LIN {X 0,Y 467.847,Z 259.021,A -85,B 0,C 180,E1 -7562.584,E2 -7562.584} C_VEL
LIN {X 0,Y 467.734,Z 259.031,A -85,B 0,C 180,E1 -7566.039,E2 -7566.039} C_VEL
LIN {X 0,Y 467.669,Z 259.046,A -85,B 0,C 180,E1 -7568.644,E2 -7568.644} C_VEL
LIN {X 0,Y 467.664,Z 259.043,A -85,B 0,C 180,E1 -7572.37,E2 -7572.37} C_VEL
LIN {X 0,Y 467.64,Z 259.045,A -85,B 0,C 180,E1 -7575.887,E2 -7575.887} C_VEL
LIN {X 0,Y 467.612,Z 259.05,A -85,B 0,C 180,E1 -7579.309,E2 -7579.309} C_VEL
LIN {X 0,Y 467.528,Z 259.059,A -85,B 0,C 180,E1 -7582.075,E2 -7582.075} C_VEL
LIN {X 0,Y 467.585,Z 259.054,A -85,B 0,C 180,E1 -7584.89,E2 -7584.89} C_VEL
LIN {X 0,Y 467.572,Z 259.059,A -85,B 0,C 180,E1 -7587.773,E2 -7587.773} C_VEL
LIN {X 0,Y 467.563,Z 259.06,A -85,B 0,C 180,E1 -7591.047,E2 -7591.047} C_VEL
LIN {X 0,Y 467.582,Z 259.057,A -85,B 0,C 180,E1 -7594.244,E2 -7594.244} C_VEL
LIN {X 0,Y 467.537,Z 259.064,A -85,B 0,C 180,E1 -7597.187,E2 -7597.187} C_VEL
LIN {X 0,Y 467.59,Z 259.056,A -85,B 0,C 180,E1 -7600.264,E2 -7600.264} C_VEL
LIN {X 0,Y 467.582,Z 259.054,A -85,B 0,C 180,E1 -7602.569,E2 -7602.569} C_VEL
LIN {X 0,Y 467.561,Z 259.062,A -85,B 0,C 180,E1 -7605.054,E2 -7605.054} C_VEL
LIN {X 0,Y 467.585,Z 259.056,A -85,B 0,C 180,E1 -7607.441,E2 -7607.441} C_VEL
LIN {X 0,Y 467.578,Z 259.057,A -85,B 0,C 180,E1 -7610.857,E2 -7610.857} C_VEL
LIN {X 0,Y 467.576,Z 259.195,A -85,B 0,C 180,E1 -7613.246,E2 -7613.246} C_VEL
LIN {X 0,Y 468.724,Z 265.645,A -85,B 0,C 180,E1 -7616.307,E2 -7616.307} C_VEL
LIN {X 0,Y 468.772,Z 270.316,A -85,B 0,C 180,E1 -7618.351,E2 -7618.351} C_VEL
LIN {X 0,Y 468.223,Z 278.68,A -85,B 0,C 180,E1 -7621.784,E2 -7621.784} C_VEL
LIN {X 0,Y 467.766,Z 287.187,A -85,B 0,C 180,E1 -7625.123,E2 -7625.123} C_VEL
LIN {X 0,Y 467.482,Z 294.551,A -85,B 0,C 180,E1 -7627.925,E2 -7627.925} C_VEL
LIN {X 0,Y 467.187,Z 304.438,A -85,B 0,C 180,E1 -7631.586,E2 -7631.586} C_VEL
LIN {X 0,Y 466.983,Z 313.335,A -85,B 0,C 180,E1 -7634.792,E2 -7634.792} C_VEL
LIN {X 0,Y 466.835,Z 321.809,A -85,B 0,C 180,E1 -7637.807,E2 -7637.807} C_VEL
LIN {X 0,Y 468.169,Z 334.234,A -85,B 0,C 180,E1 -7638.248,E2 -7638.248} C_VEL
LIN {X 0,Y 468.576,Z 341.804,A -85,B 0,C 180,E1 -7638.606,E2 -7638.606} C_VEL
LIN {X 0,Y 468.272,Z 351.549,A -85,B 0,C 180,E1 -7639.188,E2 -7639.188} C_VEL
LIN {X 0,Y 467.927,Z 360.068,A -85,B 0,C 180,E1 -7639.837,E2 -7639.837} C_VEL
LIN {X 0,Y 467.577,Z 368.103,A -85,B 0,C 180,E1 -7640.594,E2 -7640.594} C_VEL
LIN {X 0,Y 467.357,Z 374.752,A -85,B 0,C 180,E1 -7641.352,E2 -7641.352} C_VEL
LIN {X 0,Y 467.106,Z 381.074,A -85,B 0,C 180,E1 -7642.219,E2 -7642.219} C_VEL
LIN {X 0,Y 466.94,Z 386.332,A -85,B 0,C 180,E1 -7643.085,E2 -7643.085} C_VEL
LIN {X 0,Y 466.833,Z 390.722,A -85,B 0,C 180,E1 -7643.952,E2 -7643.952} C_VEL
LIN {X 0,Y 466.719,Z 395.908,A -85,B 0,C 180,E1 -7645.25,E2 -7645.25} C_VEL
LIN {X 0,Y 466.757,Z 399.722,A -85,B 0,C 180,E1 -7646.548,E2 -7646.548} C_VEL
LIN {X 0,Y 466.686,Z 401.467,A -85,B 0,C 180,E1 -7647.412,E2 -7647.412} C_VEL
LIN {X 0,Y 466.661,Z 402.717,A -85,B 0,C 180,E1 -7648.275,E2 -7648.275} C_VEL
LIN {X 0,Y 466.62,Z 403.491,A -85,B 0,C 180,E1 -7649.138,E2 -7649.138} C_VEL
LIN {X 0,Y 466.603,Z 403.785,A -85,B 0,C 180,E1 -7650.001,E2 -7650.001} C_VEL
LIN {X 0,Y 466.62,Z 403.487,A -85,B 0,C 180,E1 -7650.864,E2 -7650.864} C_VEL
LIN {X 0,Y 466.661,Z 402.692,A -85,B 0,C 180,E1 -7651.727,E2 -7651.727} C_VEL
LIN {X 0,Y 466.686,Z 401.42,A -85,B 0,C 180,E1 -7652.59,E2 -7652.59} C_VEL
LIN {X 0,Y 466.717,Z 398.486,A -85,B 0,C 180,E1 -7653.887,E2 -7653.887} C_VEL
LIN {X 0,Y 466.719,Z 395.804,A -85,B 0,C 180,E1 -7654.752,E2 -7654.752} C_VEL
LIN {X 0,Y 466.833,Z 392.504,A -85,B 0,C 180,E1 -7655.617,E2 -7655.617} C_VEL
LIN {X 0,Y 466.952,Z 387.176,A -85,B 0,C 180,E1 -7656.725,E2 -7656.725} C_VEL
LIN {X 0,Y 467.098,Z 380.806,A -85,B 0,C 180,E1 -7657.784,E2 -7657.784} C_VEL
LIN {X 0,Y 467.415,Z 372.688,A -85,B 0,C 180,E1 -7658.867,E2 -7658.867} C_VEL
LIN {X 0,Y 467.752,Z 363.177,A -85,B 0,C 180,E1 -7659.842,E2 -7659.842} C_VEL
LIN {X 0,Y 468.024,Z 355.279,A -85,B 0,C 180,E1 -7660.492,E2 -7660.492} C_VEL
LIN {X 0,Y 468.309,Z 347.164,A -85,B 0,C 180,E1 -7661.032,E2 -7661.032} C_VEL
LIN {X 0,Y 468.501,Z 338.954,A -85,B 0,C 180,E1 -7661.468,E2 -7661.468} C_VEL
LIN {X 0,Y 467.685,Z 330.12,A -85,B 0,C 180,E1 -7661.845,E2 -7661.845} C_VEL
LIN {X 0,Y 466.831,Z 321.957,A -85,B 0,C 180,E1 -7662.122,E2 -7662.122} C_VEL
LIN {X 0,Y 466.971,Z 313.201,A -85,B 0,C 180,E1 -7665.207,E2 -7665.207} C_VEL
LIN {X 0,Y 467.162,Z 304.206,A -85,B 0,C 180,E1 -7668.418,E2 -7668.418} C_VEL
LIN {X 0,Y 467.393,Z 295.384,A -85,B 0,C 180,E1 -7671.617,E2 -7671.617} C_VEL
LIN {X 0,Y 467.714,Z 286.565,A -85,B 0,C 180,E1 -7674.882,E2 -7674.882} C_VEL
LIN {X 0,Y 468.048,Z 279.032,A -85,B 0,C 180,E1 -7677.742,E2 -7677.742} C_VEL
LIN {X 0,Y 468.398,Z 271.514,A -85,B 0,C 180,E1 -7680.675,E2 -7680.675} C_VEL
LIN {X 0,Y 468.62,Z 265.139,A -85,B 0,C 180,E1 -7683.246,E2 -7683.246} C_VEL
LIN {X 0,Y 467.569,Z 259.058,A -85,B 0,C 180,E1 -7685.889,E2 -7685.889} C_VEL
LIN {X 0,Y 467.568,Z 259.057,A -85,B 0,C 180,E1 -7689.147,E2 -7689.147} C_VEL
LIN {X 0,Y 467.595,Z 259.053,A -85,B 0,C 180,E1 -7692.567,E2 -7692.567} C_VEL
LIN {X 0,Y 467.574,Z 259.054,A -85,B 0,C 180,E1 -7695.053,E2 -7695.053} C_VEL
LIN {X 0,Y 467.598,Z 259.053,A -85,B 0,C 180,E1 -7697.44,E2 -7697.44} C_VEL
LIN {X 0,Y 467.568,Z 259.056,A -85,B 0,C 180,E1 -7700.853,E2 -7700.853} C_VEL
LIN {X 0,Y 467.566,Z 259.058,A -85,B 0,C 180,E1 -7704.261,E2 -7704.261} C_VEL
LIN {X 0,Y 467.59,Z 259.055,A -85,B 0,C 180,E1 -7707.321,E2 -7707.321} C_VEL
LIN {X 0,Y 467.578,Z 259.055,A -85,B 0,C 180,E1 -7710.667,E2 -7710.667} C_VEL
LIN {X 0,Y 467.622,Z 259.051,A -85,B 0,C 180,E1 -7713.199,E2 -7713.199} C_VEL
LIN {X 0,Y 467.6,Z 259.052,A -85,B 0,C 180,E1 -7716.468,E2 -7716.468} C_VEL
LIN {X 0,Y 467.631,Z 259.048,A -85,B 0,C 180,E1 -7719.776,E2 -7719.776} C_VEL
LIN {X 0,Y 467.606,Z 259.051,A -85,B 0,C 180,E1 -7722.505,E2 -7722.505} C_VEL
LIN {X 0,Y 467.613,Z 259.052,A -85,B 0,C 180,E1 -7725.195,E2 -7725.195} C_VEL
LIN {X 0,Y 467.664,Z 259.044,A -85,B 0,C 180,E1 -7727.853,E2 -7727.853} C_VEL
LIN {X 0,Y 467.676,Z 259.043,A -85,B 0,C 180,E1 -7731.356,E2 -7731.356} C_VEL
LIN {X 0,Y 467.74,Z 259.035,A -85,B 0,C 180,E1 -7733.961,E2 -7733.961} C_VEL
LIN {X 0,Y 467.865,Z 259.019,A -85,B 0,C 180,E1 -7737.416,E2 -7737.416} C_VEL
LIN {X 0,Y 467.888,Z 259.017,A -85,B 0,C 180,E1 -7739.998,E2 -7739.998} C_VEL
LIN {X 0,Y 467.865,Z 259.021,A -85,B 0,C 180,E1 -7742.581,E2 -7742.581} C_VEL
LIN {X 0,Y 467.748,Z 259.035,A -85,B 0,C 180,E1 -7746.036,E2 -7746.036} C_VEL
LIN {X 0,Y 467.685,Z 259.043,A -85,B 0,C 180,E1 -7748.641,E2 -7748.641} C_VEL
LIN {X 0,Y 467.659,Z 259.048,A -85,B 0,C 180,E1 -7752.144,E2 -7752.144} C_VEL
LIN {X 0,Y 467.641,Z 259.048,A -85,B 0,C 180,E1 -7755.693,E2 -7755.693} C_VEL
LIN {X 0,Y 467.618,Z 259.05,A -85,B 0,C 180,E1 -7758.762,E2 -7758.762} C_VEL
LIN {X 0,Y 467.58,Z 259.055,A -85,B 0,C 180,E1 -7761.266,E2 -7761.266} C_VEL
LIN {X 0,Y 467.572,Z 259.057,A -85,B 0,C 180,E1 -7763.941,E2 -7763.941} C_VEL
LIN {X 0,Y 467.614,Z 259.049,A -85,B 0,C 180,E1 -7766.798,E2 -7766.798} C_VEL
LIN {X 0,Y 467.551,Z 259.06,A -85,B 0,C 180,E1 -7769.736,E2 -7769.736} C_VEL
LIN {X 0,Y 467.58,Z 259.054,A -85,B 0,C 180,E1 -7772.756,E2 -7772.756} C_VEL
LIN {X 0,Y 467.551,Z 259.059,A -85,B 0,C 180,E1 -7775.887,E2 -7775.887} C_VEL
LIN {X 0,Y 467.608,Z 259.052,A -85,B 0,C 180,E1 -7779.139,E2 -7779.139} C_VEL
LIN {X 0,Y 467.611,Z 259.051,A -85,B 0,C 180,E1 -7782.569,E2 -7782.569} C_VEL
LIN {X 0,Y 467.565,Z 259.056,A -85,B 0,C 180,E1 -7786.174,E2 -7786.174} C_VEL
LIN {X 0,Y 467.581,Z 259.057,A -85,B 0,C 180,E1 -7788.719,E2 -7788.719} C_VEL
LIN {X 0,Y 467.568,Z 259.058,A -85,B 0,C 180,E1 -7791.404,E2 -7791.404} C_VEL
LIN {X 0,Y 467.552,Z 259.057,A -85,B 0,C 180,E1 -7794.258,E2 -7794.258} C_VEL
LIN {X 0,Y 467.569,Z 259.058,A -85,B 0,C 180,E1 -7797.319,E2 -7797.319} C_VEL
LIN {X 0,Y 467.564,Z 259.059,A -85,B 0,C 180,E1 -7800.663,E2 -7800.663} C_VEL
LIN {X 0,Y 467.613,Z 259.051,A -85,B 0,C 180,E1 -7803.198,E2 -7803.198} C_VEL
LIN {X 0,Y 467.582,Z 259.056,A -85,B 0,C 180,E1 -7806.465,E2 -7806.465} C_VEL
LIN {X 0,Y 467.603,Z 259.052,A -85,B 0,C 180,E1 -7809.775,E2 -7809.775} C_VEL
LIN {X 0,Y 467.545,Z 259.059,A -85,B 0,C 180,E1 -7811.629,E2 -7811.629} C_VEL
LIN {X 0,Y 467.186,Z 259.106,A -85,B 0,C 180,E1 -7814.306,E2 -7814.306} C_VEL
LIN {X 0,Y 467.136,Z 260.347,A -85,B 0,C 180,E1 -7815.376,E2 -7815.376} C_VEL
LIN {X 0,Y 466.444,Z 261.32,A -85,B 0,C 180,E1 -7816.087,E2 -7816.087} C_VEL
LIN {X 0,Y 463.58,Z 263.063,A -85,B 0,C 180,E1 -7817.238,E2 -7817.238} C_VEL
LIN {X 0,Y 461.159,Z 264.477,A -85,B 0,C 180,E1 -7818.166,E2 -7818.166} C_VEL
LIN {X 0,Y 460.102,Z 265.496,A -85,B 0,C 180,E1 -7818.884,E2 -7818.884} C_VEL
LIN {X 0,Y 460.005,Z 265.819,A -85,B 0,C 180,E1 -7819.127,E2 -7819.127} C_VEL
LIN {X 0,Y 459.965,Z 269.626,A -85,B 0,C 180,E1 -7822.095,E2 -7822.095} C_VEL
LIN {X 0,Y 459.987,Z 271.938,A -85,B 0,C 180,E1 -7823.859,E2 -7823.859} C_VEL
LIN {X 0,Y 459.964,Z 275.389,A -85,B 0,C 180,E1 -7826.495,E2 -7826.495} C_VEL
LIN {X 0,Y 459.636,Z 280.076,A -85,B 0,C 180,E1 -7829.999,E2 -7829.999} C_VEL
LIN {X 0,Y 459.646,Z 282.543,A -85,B 0,C 180,E1 -7831.833,E2 -7831.833} C_VEL
LIN {X 0,Y 461.767,Z 294.466,A -85,B 0,C 180,E1 -7832.343,E2 -7832.343} C_VEL
LIN {X 0,Y 461.645,Z 302.062,A -85,B 0,C 180,E1 -7832.726,E2 -7832.726} C_VEL
LIN {X 0,Y 461.4,Z 310.62,A -85,B 0,C 180,E1 -7833.273,E2 -7833.273} C_VEL
LIN {X 0,Y 461.077,Z 318.847,A -85,B 0,C 180,E1 -7833.932,E2 -7833.932} C_VEL
LIN {X 0,Y 460.768,Z 326.642,A -85,B 0,C 180,E1 -7834.701,E2 -7834.701} C_VEL
LIN {X 0,Y 460.59,Z 333.057,A -85,B 0,C 180,E1 -7835.471,E2 -7835.471} C_VEL
LIN {X 0,Y 460.357,Z 338.967,A -85,B 0,C 180,E1 -7836.319,E2 -7836.319} C_VEL
LIN {X 0,Y 460.201,Z 344.276,A -85,B 0,C 180,E1 -7837.237,E2 -7837.237} C_VEL
LIN {X 0,Y 459.932,Z 349.496,A -85,B 0,C 180,E1 -7838.346,E2 -7838.346} C_VEL
LIN {X 0,Y 459.757,Z 354.317,A -85,B 0,C 180,E1 -7839.679,E2 -7839.679} C_VEL
LIN {X 0,Y 459.698,Z 356.67,A -85,B 0,C 180,E1 -7840.57,E2 -7840.57} C_VEL
LIN {X 0,Y 459.63,Z 359.185,A -85,B 0,C 180,E1 -7841.89,E2 -7841.89} C_VEL
LIN {X 0,Y 459.534,Z 360.484,A -85,B 0,C 180,E1 -7843.261,E2 -7843.261} C_VEL
LIN {X 0,Y 459.507,Z 360.759,A -85,B 0,C 180,E1 -7844.164,E2 -7844.164} C_VEL
LIN {X 0,Y 459.581,Z 360.016,A -85,B 0,C 180,E1 -7845.558,E2 -7845.558} C_VEL
LIN {X 0,Y 459.654,Z 358.169,A -85,B 0,C 180,E1 -7846.887,E2 -7846.887} C_VEL
LIN {X 0,Y 459.781,Z 355.119,A -85,B 0,C 180,E1 -7848.225,E2 -7848.225} C_VEL
LIN {X 0,Y 460.03,Z 350.431,A -85,B 0,C 180,E1 -7849.638,E2 -7849.638} C_VEL
LIN {X 0,Y 460.2,Z 345.355,A -85,B 0,C 180,E1 -7850.767,E2 -7850.767} C_VEL
LIN {X 0,Y 460.429,Z 340.034,A -85,B 0,C 180,E1 -7851.724,E2 -7851.724} C_VEL
LIN {X 0,Y 460.7,Z 333.714,A -85,B 0,C 180,E1 -7852.654,E2 -7852.654} C_VEL
LIN {X 0,Y 460.98,Z 326.74,A -85,B 0,C 180,E1 -7853.499,E2 -7853.499} C_VEL
LIN {X 0,Y 461.303,Z 318.786,A -85,B 0,C 180,E1 -7854.288,E2 -7854.288} C_VEL
LIN {X 0,Y 461.701,Z 310.029,A -85,B 0,C 180,E1 -7854.985,E2 -7854.985} C_VEL
LIN {X 0,Y 462.023,Z 299.473,A -85,B 0,C 180,E1 -7855.639,E2 -7855.639} C_VEL
LIN {X 0,Y 461.889,Z 294.564,A -85,B 0,C 180,E1 -7855.875,E2 -7855.875} C_VEL
LIN {X 0,Y 460.037,Z 284.59,A -85,B 0,C 180,E1 -7856.316,E2 -7856.316} C_VEL
LIN {X 0,Y 459.668,Z 282.744,A -85,B 0,C 180,E1 -7856.395,E2 -7856.395} C_VEL
LIN {X 0,Y 459.727,Z 278.823,A -85,B 0,C 180,E1 -7859.386,E2 -7859.386} C_VEL
LIN {X 0,Y 459.793,Z 275.013,A -85,B 0,C 180,E1 -7862.341,E2 -7862.341} C_VEL
LIN {X 0,Y 459.887,Z 270.511,A -85,B 0,C 180,E1 -7865.914,E2 -7865.914} C_VEL
LIN {X 0,Y 459.949,Z 266.915,A -85,B 0,C 180,E1 -7868.809,E2 -7868.809} C_VEL
LIN {X 0,Y 460.094,Z 262.754,A -85,B 0,C 180,E1 -7872.228,E2 -7872.228} C_VEL
LIN {X 0,Y 460.179,Z 259.979,A -85,B 0,C 180,E1 -7874.628,E2 -7874.628} C_VEL
LIN {X 0,Y 460.412,Z 259.944,A -85,B 0,C 180,E1 -7877.111,E2 -7877.111} C_VEL
LIN {X 0,Y 460.557,Z 259.928,A -85,B 0,C 180,E1 -7880.143,E2 -7880.143} C_VEL
LIN {X 0,Y 460.461,Z 259.941,A -85,B 0,C 180,E1 -7883.472,E2 -7883.472} C_VEL
LIN {X 0,Y 460.51,Z 259.934,A -85,B 0,C 180,E1 -7886.676,E2 -7886.676} C_VEL
LIN {X 0,Y 460.491,Z 259.936,A -85,B 0,C 180,E1 -7889.761,E2 -7889.761} C_VEL
LIN {X 0,Y 460.56,Z 259.927,A -85,B 0,C 180,E1 -7892.758,E2 -7892.758} C_VEL
LIN {X 0,Y 460.52,Z 259.932,A -85,B 0,C 180,E1 -7895.669,E2 -7895.669} C_VEL
LIN {X 0,Y 460.504,Z 259.936,A -85,B 0,C 180,E1 -7898.579,E2 -7898.579} C_VEL
LIN {X 0,Y 460.575,Z 259.927,A -85,B 0,C 180,E1 -7901.312,E2 -7901.312} C_VEL
LIN {X 0,Y 460.588,Z 259.924,A -85,B 0,C 180,E1 -7904.06,E2 -7904.06} C_VEL
LIN {X 0,Y 460.615,Z 259.922,A -85,B 0,C 180,E1 -7907.668,E2 -7907.668} C_VEL
LIN {X 0,Y 460.615,Z 259.925,A -85,B 0,C 180,E1 -7911.225,E2 -7911.225} C_VEL
LIN {X 0,Y 460.671,Z 259.911,A -85,B 0,C 180,E1 -7913.871,E2 -7913.871} C_VEL
LIN {X 0,Y 460.815,Z 259.898,A -85,B 0,C 180,E1 -7917.379,E2 -7917.379} C_VEL
LIN {X 0,Y 460.84,Z 259.892,A -85,B 0,C 180,E1 -7920.002,E2 -7920.002} C_VEL
LIN {X 0,Y 460.788,Z 259.9,A -85,B 0,C 180,E1 -7922.624,E2 -7922.624} C_VEL
LIN {X 0,Y 460.7,Z 259.906,A -85,B 0,C 180,E1 -7926.131,E2 -7926.131} C_VEL
LIN {X 0,Y 460.616,Z 259.923,A -85,B 0,C 180,E1 -7928.778,E2 -7928.778} C_VEL
LIN {X 0,Y 460.625,Z 259.919,A -85,B 0,C 180,E1 -7932.458,E2 -7932.458} C_VEL
LIN {X 0,Y 460.591,Z 259.924,A -85,B 0,C 180,E1 -7935.999,E2 -7935.999} C_VEL
LIN {X 0,Y 460.559,Z 259.931,A -85,B 0,C 180,E1 -7939.617,E2 -7939.617} C_VEL
LIN {X 0,Y 460.504,Z 259.935,A -85,B 0,C 180,E1 -7942.43,E2 -7942.43} C_VEL
LIN {X 0,Y 460.542,Z 259.933,A -85,B 0,C 180,E1 -7945.799,E2 -7945.799} C_VEL
LIN {X 0,Y 460.519,Z 259.934,A -85,B 0,C 180,E1 -7948.236,E2 -7948.236} C_VEL
LIN {X 0,Y 460.516,Z 259.936,A -85,B 0,C 180,E1 -7951.285,E2 -7951.285} C_VEL
LIN {X 0,Y 460.525,Z 259.935,A -85,B 0,C 180,E1 -7954.507,E2 -7954.507} C_VEL
LIN {X 0,Y 460.495,Z 259.937,A -85,B 0,C 180,E1 -7957.625,E2 -7957.625} C_VEL
LIN {X 0,Y 460.553,Z 259.933,A -85,B 0,C 180,E1 -7960.273,E2 -7960.273} C_VEL
LIN {X 0,Y 460.494,Z 259.941,A -85,B 0,C 180,E1 -7963.377,E2 -7963.377} C_VEL
LIN {X 0,Y 460.494,Z 259.938,A -85,B 0,C 180,E1 -7966.626,E2 -7966.626} C_VEL
LIN {X 0,Y 460.538,Z 259.934,A -85,B 0,C 180,E1 -7969.732,E2 -7969.732} C_VEL
LIN {X 0,Y 460.508,Z 259.977,A -85,B 0,C 180,E1 -7972.929,E2 -7972.929} C_VEL
LIN {X 0,Y 461.544,Z 265.68,A -85,B 0,C 180,E1 -7975.71,E2 -7975.71} C_VEL
LIN {X 0,Y 461.861,Z 269.21,A -85,B 0,C 180,E1 -7977.325,E2 -7977.325} C_VEL
LIN {X 0,Y 461.446,Z 276.023,A -85,B 0,C 180,E1 -7980.243,E2 -7980.243} C_VEL
LIN {X 0,Y 460.978,Z 283.444,A -85,B 0,C 180,E1 -7983.274,E2 -7983.274} C_VEL
LIN {X 0,Y 460.581,Z 291.954,A -85,B 0,C 180,E1 -7986.627,E2 -7986.627} C_VEL
LIN {X 0,Y 460.207,Z 300.556,A -85,B 0,C 180,E1 -7989.905,E2 -7989.905} C_VEL
LIN {X 0,Y 459.993,Z 309.209,A -85,B 0,C 180,E1 -7993.126,E2 -7993.126} C_VEL
LIN {X 0,Y 459.8,Z 317.907,A -85,B 0,C 180,E1 -7996.297,E2 -7996.297} C_VEL
LIN {X 0,Y 459.762,Z 321.484,A -85,B 0,C 180,E1 -7997.588,E2 -7997.588} C_VEL
LIN {X 0,Y 461.195,Z 334.661,A -85,B 0,C 180,E1 -7998.082,E2 -7998.082} C_VEL
LIN {X 0,Y 461.623,Z 342.117,A -85,B 0,C 180,E1 -7998.448,E2 -7998.448} C_VEL
LIN {X 0,Y 461.308,Z 351.464,A -85,B 0,C 180,E1 -7999.023,E2 -7999.023} C_VEL
LIN {X 0,Y 460.935,Z 359.927,A -85,B 0,C 180,E1 -7999.681,E2 -7999.681} C_VEL
LIN {X 0,Y 460.564,Z 367.92,A -85,B 0,C 180,E1 -8000.449,E2 -8000.449} C_VEL
LIN {X 0,Y 460.306,Z 374.536,A -85,B 0,C 180,E1 -8001.219,E2 -8001.219} C_VEL
LIN {X 0,Y 460.062,Z 380.831,A -85,B 0,C 180,E1 -8002.099,E2 -8002.099} C_VEL
LIN {X 0,Y 459.873,Z 386.07,A -85,B 0,C 180,E1 -8002.979,E2 -8002.979} C_VEL
LIN {X 0,Y 459.742,Z 390.446,A -85,B 0,C 180,E1 -8003.858,E2 -8003.858} C_VEL
LIN {X 0,Y 459.65,Z 395.622,A -85,B 0,C 180,E1 -8005.177,E2 -8005.177} C_VEL
LIN {X 0,Y 459.651,Z 399.424,A -85,B 0,C 180,E1 -8006.495,E2 -8006.495} C_VEL
LIN {X 0,Y 459.609,Z 401.161,A -85,B 0,C 180,E1 -8007.372,E2 -8007.372} C_VEL
LIN {X 0,Y 459.57,Z 402.401,A -85,B 0,C 180,E1 -8008.248,E2 -8008.248} C_VEL
LIN {X 0,Y 459.553,Z 403.167,A -85,B 0,C 180,E1 -8009.125,E2 -8009.125} C_VEL
LIN {X 0,Y 459.534,Z 403.455,A -85,B 0,C 180,E1 -8010.001,E2 -8010.001} C_VEL
LIN {X 0,Y 459.553,Z 403.154,A -85,B 0,C 180,E1 -8010.877,E2 -8010.877} C_VEL
LIN {X 0,Y 459.571,Z 402.348,A -85,B 0,C 180,E1 -8011.754,E2 -8011.754} C_VEL
LIN {X 0,Y 459.609,Z 401.066,A -85,B 0,C 180,E1 -8012.63,E2 -8012.63} C_VEL
LIN {X 0,Y 459.611,Z 398.119,A -85,B 0,C 180,E1 -8013.947,E2 -8013.947} C_VEL
LIN {X 0,Y 459.651,Z 395.427,A -85,B 0,C 180,E1 -8014.825,E2 -8014.825} C_VEL
LIN {X 0,Y 459.732,Z 392.113,A -85,B 0,C 180,E1 -8015.704,E2 -8015.704} C_VEL
LIN {X 0,Y 459.883,Z 387.077,A -85,B 0,C 180,E1 -8016.772,E2 -8016.772} C_VEL
LIN {X 0,Y 459.993,Z 381.813,A -85,B 0,C 180,E1 -8017.684,E2 -8017.684} C_VEL
LIN {X 0,Y 460.224,Z 375.68,A -85,B 0,C 180,E1 -8018.564,E2 -8018.564} C_VEL
LIN {X 0,Y 460.446,Z 369.243,A -85,B 0,C 180,E1 -8019.334,E2 -8019.334} C_VEL
LIN {X 0,Y 460.786,Z 361.452,A -85,B 0,C 180,E1 -8020.103,E2 -8020.103} C_VEL
LIN {X 0,Y 461.023,Z 354.747,A -85,B 0,C 180,E1 -8020.653,E2 -8020.653} C_VEL
LIN {X 0,Y 461.314,Z 346.571,A -85,B 0,C 180,E1 -8021.202,E2 -8021.202} C_VEL
LIN {X 0,Y 461.434,Z 338.943,A -85,B 0,C 180,E1 -8021.614,E2 -8021.614} C_VEL
LIN {X 0,Y 460.547,Z 329.166,A -85,B 0,C 180,E1 -8022.033,E2 -8022.033} C_VEL
LIN {X 0,Y 459.752,Z 321.703,A -85,B 0,C 180,E1 -8022.275,E2 -8022.275} C_VEL
LIN {X 0,Y 459.921,Z 312.172,A -85,B 0,C 180,E1 -8025.698,E2 -8025.698} C_VEL
LIN {X 0,Y 460.115,Z 302.765,A -85,B 0,C 180,E1 -8029.126,E2 -8029.126} C_VEL
LIN {X 0,Y 460.408,Z 293.823,A -85,B 0,C 180,E1 -8032.435,E2 -8032.435} C_VEL
LIN {X 0,Y 460.773,Z 284.821,A -85,B 0,C 180,E1 -8035.853,E2 -8035.853} C_VEL
LIN {X 0,Y 461.18,Z 276.269,A -85,B 0,C 180,E1 -8039.187,E2 -8039.187} C_VEL
LIN {X 0,Y 461.566,Z 268.781,A -85,B 0,C 180,E1 -8042.204,E2 -8042.204} C_VEL
LIN {X 0,Y 461.442,Z 265.042,A -85,B 0,C 180,E1 -8043.775,E2 -8043.775} C_VEL
LIN {X 0,Y 460.507,Z 259.938,A -85,B 0,C 180,E1 -8046.089,E2 -8046.089} C_VEL
LIN {X 0,Y 460.542,Z 259.932,A -85,B 0,C 180,E1 -8048.896,E2 -8048.896} C_VEL
LIN {X 0,Y 460.531,Z 259.935,A -85,B 0,C 180,E1 -8052.182,E2 -8052.182} C_VEL
LIN {X 0,Y 460.521,Z 259.934,A -85,B 0,C 180,E1 -8055.411,E2 -8055.411} C_VEL
LIN {X 0,Y 460.54,Z 259.932,A -85,B 0,C 180,E1 -8058.398,E2 -8058.398} C_VEL
LIN {X 0,Y 460.526,Z 259.934,A -85,B 0,C 180,E1 -8061.266,E2 -8061.266} C_VEL
LIN {X 0,Y 460.517,Z 259.934,A -85,B 0,C 180,E1 -8064.554,E2 -8064.554} C_VEL
LIN {X 0,Y 460.54,Z 259.933,A -85,B 0,C 180,E1 -8067.715,E2 -8067.715} C_VEL
LIN {X 0,Y 460.548,Z 259.931,A -85,B 0,C 180,E1 -8070.768,E2 -8070.768} C_VEL
LIN {X 0,Y 460.565,Z 259.93,A -85,B 0,C 180,E1 -8073.734,E2 -8073.734} C_VEL
LIN {X 0,Y 460.553,Z 259.93,A -85,B 0,C 180,E1 -8076.623,E2 -8076.623} C_VEL
LIN {X 0,Y 460.56,Z 259.931,A -85,B 0,C 180,E1 -8079.452,E2 -8079.452} C_VEL
LIN {X 0,Y 460.557,Z 259.928,A -85,B 0,C 180,E1 -8082.229,E2 -8082.229} C_VEL
LIN {X 0,Y 460.572,Z 259.93,A -85,B 0,C 180,E1 -8084.964,E2 -8084.964} C_VEL
LIN {X 0,Y 460.617,Z 259.923,A -85,B 0,C 180,E1 -8088.558,E2 -8088.558} C_VEL
LIN {X 0,Y 460.626,Z 259.922,A -85,B 0,C 180,E1 -8091.222,E2 -8091.222} C_VEL
LIN {X 0,Y 460.705,Z 259.911,A -85,B 0,C 180,E1 -8093.869,E2 -8093.869} C_VEL
LIN {X 0,Y 460.806,Z 259.898,A -85,B 0,C 180,E1 -8097.376,E2 -8097.376} C_VEL
LIN {X 0,Y 460.858,Z 259.892,A -85,B 0,C 180,E1 -8099.998,E2 -8099.998} C_VEL
LIN {X 0,Y 460.83,Z 259.897,A -85,B 0,C 180,E1 -8102.621,E2 -8102.621} C_VEL
LIN {X 0,Y 460.714,Z 259.912,A -85,B 0,C 180,E1 -8106.128,E2 -8106.128} C_VEL
LIN {X 0,Y 460.632,Z 259.922,A -85,B 0,C 180,E1 -8108.774,E2 -8108.774} C_VEL
LIN {X 0,Y 460.616,Z 259.923,A -85,B 0,C 180,E1 -8112.443,E2 -8112.443} C_VEL
LIN {X 0,Y 460.602,Z 259.926,A -85,B 0,C 180,E1 -8115.995,E2 -8115.995} C_VEL
LIN {X 0,Y 460.572,Z 259.928,A -85,B 0,C 180,E1 -8118.9,E2 -8118.9} C_VEL
LIN {X 0,Y 460.516,Z 259.936,A -85,B 0,C 180,E1 -8121.483,E2 -8121.483} C_VEL
LIN {X 0,Y 460.541,Z 259.932,A -85,B 0,C 180,E1 -8124.33,E2 -8124.33} C_VEL
LIN {X 0,Y 460.577,Z 259.927,A -85,B 0,C 180,E1 -8127.241,E2 -8127.241} C_VEL
LIN {X 0,Y 460.508,Z 259.936,A -85,B 0,C 180,E1 -8130.238,E2 -8130.238} C_VEL
LIN {X 0,Y 460.525,Z 259.935,A -85,B 0,C 180,E1 -8133.323,E2 -8133.323} C_VEL
LIN {X 0,Y 460.473,Z 259.939,A -85,B 0,C 180,E1 -8136.527,E2 -8136.527} C_VEL
LIN {X 0,Y 460.569,Z 259.929,A -85,B 0,C 180,E1 -8139.855,E2 -8139.855} C_VEL
LIN {X 0,Y 460.535,Z 259.933,A -85,B 0,C 180,E1 -8142.902,E2 -8142.902} C_VEL
LIN {X 0,Y 460.515,Z 259.935,A -85,B 0,C 180,E1 -8145.826,E2 -8145.826} C_VEL
LIN {X 0,Y 460.534,Z 259.934,A -85,B 0,C 180,E1 -8148.988,E2 -8148.988} C_VEL
LIN {X 0,Y 460.537,Z 259.934,A -85,B 0,C 180,E1 -8151.267,E2 -8151.267} C_VEL
LIN {X 0,Y 460.502,Z 259.937,A -85,B 0,C 180,E1 -8154.553,E2 -8154.553} C_VEL
LIN {X 0,Y 460.52,Z 259.934,A -85,B 0,C 180,E1 -8157.714,E2 -8157.714} C_VEL
LIN {X 0,Y 460.534,Z 259.935,A -85,B 0,C 180,E1 -8160.768,E2 -8160.768} C_VEL
LIN {X 0,Y 460.553,Z 259.93,A -85,B 0,C 180,E1 -8163.733,E2 -8163.733} C_VEL
LIN {X 0,Y 460.536,Z 259.935,A -85,B 0,C 180,E1 -8166.622,E2 -8166.622} C_VEL
LIN {X 0,Y 460.552,Z 259.93,A -85,B 0,C 180,E1 -8169.452,E2 -8169.452} C_VEL
LIN {X 0,Y 460.377,Z 259.954,A -85,B 0,C 180,E1 -8172.222,E2 -8172.222} C_VEL
LIN {X 0,Y 460.146,Z 259.983,A -85,B 0,C 180,E1 -8174.192,E2 -8174.192} C_VEL
LIN {X 0,Y 460.066,Z 261.03,A -85,B 0,C 180,E1 -8175.357,E2 -8175.357} C_VEL
LIN {X 0,Y 460.137,Z 264.123,A -85,B 0,C 180,E1 -8177.815,E2 -8177.815} C_VEL
LIN {X 0,Y 460.005,Z 265.819,A -85,B 0,C 180,E1 -8179.127,E2 -8179.127} C_VEL
LIN {X 0,Y 459.305,Z 266.814,A -85,B 0,C 180,E1 -8179.847,E2 -8179.847} C_VEL
LIN {X 0,Y 456.424,Z 268.581,A -85,B 0,C 180,E1 -8181.013,E2 -8181.013} C_VEL
LIN {X 0,Y 454.022,Z 270.002,A -85,B 0,C 180,E1 -8181.953,E2 -8181.953} C_VEL
LIN {X 0,Y 453.016,Z 271.021,A -85,B 0,C 180,E1 -8182.681,E2 -8182.681} C_VEL
LIN {X 0,Y 452.946,Z 271.343,A -85,B 0,C 180,E1 -8182.928,E2 -8182.928} C_VEL
LIN {X 0,Y 452.886,Z 275.91,A -85,B 0,C 180,E1 -8186.44,E2 -8186.44} C_VEL
LIN {X 0,Y 452.562,Z 280.628,A -85,B 0,C 180,E1 -8189.999,E2 -8189.999} C_VEL
LIN {X 0,Y 452.579,Z 282.861,A -85,B 0,C 180,E1 -8191.667,E2 -8191.667} C_VEL
LIN {X 0,Y 454.63,Z 294.343,A -85,B 0,C 180,E1 -8192.158,E2 -8192.158} C_VEL
LIN {X 0,Y 454.733,Z 300.061,A -85,B 0,C 180,E1 -8192.435,E2 -8192.435} C_VEL
LIN {X 0,Y 454.425,Z 310.592,A -85,B 0,C 180,E1 -8193.102,E2 -8193.102} C_VEL
LIN {X 0,Y 454.112,Z 318.874,A -85,B 0,C 180,E1 -8193.77,E2 -8193.77} C_VEL
LIN {X 0,Y 453.775,Z 326.722,A -85,B 0,C 180,E1 -8194.551,E2 -8194.551} C_VEL
LIN {X 0,Y 453.57,Z 333.182,A -85,B 0,C 180,E1 -8195.333,E2 -8195.333} C_VEL
LIN {X 0,Y 453.299,Z 339.352,A -85,B 0,C 180,E1 -8196.229,E2 -8196.229} C_VEL
LIN {X 0,Y 453.102,Z 345.643,A -85,B 0,C 180,E1 -8197.351,E2 -8197.351} C_VEL
LIN {X 0,Y 452.845,Z 350.67,A -85,B 0,C 180,E1 -8198.477,E2 -8198.477} C_VEL
LIN {X 0,Y 452.657,Z 355.183,A -85,B 0,C 180,E1 -8199.832,E2 -8199.832} C_VEL
LIN {X 0,Y 452.617,Z 357.476,A -85,B 0,C 180,E1 -8200.737,E2 -8200.737} C_VEL
LIN {X 0,Y 452.545,Z 359.599,A -85,B 0,C 180,E1 -8201.947,E2 -8201.947} C_VEL
LIN {X 0,Y 452.429,Z 360.888,A -85,B 0,C 180,E1 -8203.473,E2 -8203.473} C_VEL
LIN {X 0,Y 452.44,Z 361.022,A -85,B 0,C 180,E1 -8204.39,E2 -8204.39} C_VEL
LIN {X 0,Y 452.492,Z 360.297,A -85,B 0,C 180,E1 -8205.651,E2 -8205.651} C_VEL
LIN {X 0,Y 452.53,Z 359.679,A -85,B 0,C 180,E1 -8206.232,E2 -8206.232} C_VEL
LIN {X 0,Y 452.667,Z 357.212,A -85,B 0,C 180,E1 -8207.622,E2 -8207.622} C_VEL
LIN {X 0,Y 452.831,Z 353.298,A -85,B 0,C 180,E1 -8209.02,E2 -8209.02} C_VEL
LIN {X 0,Y 453.007,Z 349.884,A -85,B 0,C 180,E1 -8209.955,E2 -8209.955} C_VEL
LIN {X 0,Y 453.181,Z 345.676,A -85,B 0,C 180,E1 -8210.895,E2 -8210.895} C_VEL
LIN {X 0,Y 453.415,Z 340.537,A -85,B 0,C 180,E1 -8211.838,E2 -8211.838} C_VEL
LIN {X 0,Y 453.694,Z 334.25,A -85,B 0,C 180,E1 -8212.783,E2 -8212.783} C_VEL
LIN {X 0,Y 453.997,Z 327.583,A -85,B 0,C 180,E1 -8213.611,E2 -8213.611} C_VEL
LIN {X 0,Y 454.333,Z 319.976,A -85,B 0,C 180,E1 -8214.39,E2 -8214.39} C_VEL
LIN {X 0,Y 454.699,Z 312.311,A -85,B 0,C 180,E1 -8215.03,E2 -8215.03} C_VEL
LIN {X 0,Y 455.004,Z 303.475,A -85,B 0,C 180,E1 -8215.624,E2 -8215.624} C_VEL
LIN {X 0,Y 455,Z 295.645,A -85,B 0,C 180,E1 -8216.044,E2 -8216.044} C_VEL
LIN {X 0,Y 453.257,Z 286.337,A -85,B 0,C 180,E1 -8216.479,E2 -8216.479} C_VEL
LIN {X 0,Y 452.596,Z 283.071,A -85,B 0,C 180,E1 -8216.634,E2 -8216.634} C_VEL
LIN {X 0,Y 452.66,Z 278.969,A -85,B 0,C 180,E1 -8219.789,E2 -8219.789} C_VEL
LIN {X 0,Y 452.744,Z 274.813,A -85,B 0,C 180,E1 -8223.049,E2 -8223.049} C_VEL
LIN {X 0,Y 452.819,Z 270.898,A -85,B 0,C 180,E1 -8226.194,E2 -8226.194} C_VEL
LIN {X 0,Y 452.904,Z 266.851,A -85,B 0,C 180,E1 -8229.509,E2 -8229.509} C_VEL
LIN {X 0,Y 453.011,Z 264.005,A -85,B 0,C 180,E1 -8231.873,E2 -8231.873} C_VEL
LIN {X 0,Y 453.113,Z 260.92,A -85,B 0,C 180,E1 -8234.485,E2 -8234.485} C_VEL
LIN {X 0,Y 453.355,Z 260.824,A -85,B 0,C 180,E1 -8236.996,E2 -8236.996} C_VEL
LIN {X 0,Y 453.495,Z 260.811,A -85,B 0,C 180,E1 -8239.407,E2 -8239.407} C_VEL
LIN {X 0,Y 453.458,Z 260.814,A -85,B 0,C 180,E1 -8242.223,E2 -8242.223} C_VEL
LIN {X 0,Y 453.47,Z 260.812,A -85,B 0,C 180,E1 -8245.223,E2 -8245.223} C_VEL
LIN {X 0,Y 453.446,Z 260.814,A -85,B 0,C 180,E1 -8248.476,E2 -8248.476} C_VEL
LIN {X 0,Y 453.519,Z 260.807,A -85,B 0,C 180,E1 -8252.04,E2 -8252.04} C_VEL
LIN {X 0,Y 453.489,Z 260.812,A -85,B 0,C 180,E1 -8255.266,E2 -8255.266} C_VEL
LIN {X 0,Y 453.463,Z 260.815,A -85,B 0,C 180,E1 -8258.416,E2 -8258.416} C_VEL
LIN {X 0,Y 453.506,Z 260.806,A -85,B 0,C 180,E1 -8261.01,E2 -8261.01} C_VEL
LIN {X 0,Y 453.553,Z 260.8,A -85,B 0,C 180,E1 -8263.881,E2 -8263.881} C_VEL
LIN {X 0,Y 453.587,Z 260.796,A -85,B 0,C 180,E1 -8267.474,E2 -8267.474} C_VEL
LIN {X 0,Y 453.579,Z 260.799,A -85,B 0,C 180,E1 -8271.088,E2 -8271.088} C_VEL
LIN {X 0,Y 453.636,Z 260.787,A -85,B 0,C 180,E1 -8273.776,E2 -8273.776} C_VEL
LIN {X 0,Y 453.756,Z 260.777,A -85,B 0,C 180,E1 -8277.338,E2 -8277.338} C_VEL
LIN {X 0,Y 453.81,Z 260.768,A -85,B 0,C 180,E1 -8280.002,E2 -8280.002} C_VEL
LIN {X 0,Y 453.732,Z 260.778,A -85,B 0,C 180,E1 -8282.665,E2 -8282.665} C_VEL
LIN {X 0,Y 453.668,Z 260.782,A -85,B 0,C 180,E1 -8286.227,E2 -8286.227} C_VEL
LIN {X 0,Y 453.58,Z 260.798,A -85,B 0,C 180,E1 -8288.915,E2 -8288.915} C_VEL
LIN {X 0,Y 453.593,Z 260.795,A -85,B 0,C 180,E1 -8292.552,E2 -8292.552} C_VEL
LIN {X 0,Y 453.535,Z 260.804,A -85,B 0,C 180,E1 -8296.198,E2 -8296.198} C_VEL
LIN {X 0,Y 453.508,Z 260.806,A -85,B 0,C 180,E1 -8299.041,E2 -8299.041} C_VEL
LIN {X 0,Y 453.469,Z 260.811,A -85,B 0,C 180,E1 -8301.838,E2 -8301.838} C_VEL
LIN {X 0,Y 453.498,Z 260.81,A -85,B 0,C 180,E1 -8304.737,E2 -8304.737} C_VEL
LIN {X 0,Y 453.499,Z 260.81,A -85,B 0,C 180,E1 -8307.955,E2 -8307.955} C_VEL
LIN {X 0,Y 453.469,Z 260.818,A -85,B 0,C 180,E1 -8310.761,E2 -8310.761} C_VEL
LIN {X 0,Y 453.47,Z 260.817,A -85,B 0,C 180,E1 -8313.914,E2 -8313.914} C_VEL
LIN {X 0,Y 453.444,Z 260.819,A -85,B 0,C 180,E1 -8317.192,E2 -8317.192} C_VEL
LIN {X 0,Y 453.526,Z 260.805,A -85,B 0,C 180,E1 -8319.447,E2 -8319.447} C_VEL
LIN {X 0,Y 453.458,Z 260.814,A -85,B 0,C 180,E1 -8322.997,E2 -8322.997} C_VEL
LIN {X 0,Y 453.459,Z 260.813,A -85,B 0,C 180,E1 -8325.78,E2 -8325.78} C_VEL
LIN {X 0,Y 453.476,Z 260.815,A -85,B 0,C 180,E1 -8328.211,E2 -8328.211} C_VEL
LIN {X 0,Y 453.491,Z 260.812,A -85,B 0,C 180,E1 -8330.795,E2 -8330.795} C_VEL
LIN {X 0,Y 453.461,Z 260.897,A -85,B 0,C 180,E1 -8332.668,E2 -8332.668} C_VEL
LIN {X 0,Y 454.574,Z 266.903,A -85,B 0,C 180,E1 -8335.647,E2 -8335.647} C_VEL
LIN {X 0,Y 454.879,Z 270.323,A -85,B 0,C 180,E1 -8337.266,E2 -8337.266} C_VEL
LIN {X 0,Y 454.46,Z 276.625,A -85,B 0,C 180,E1 -8340,E2 -8340} C_VEL
LIN {X 0,Y 453.985,Z 283.396,A -85,B 0,C 180,E1 -8342.828,E2 -8342.828} C_VEL
LIN {X 0,Y 453.551,Z 291.843,A -85,B 0,C 180,E1 -8346.243,E2 -8346.243} C_VEL
LIN {X 0,Y 453.184,Z 300.398,A -85,B 0,C 180,E1 -8349.579,E2 -8349.579} C_VEL
LIN {X 0,Y 452.915,Z 309.026,A -85,B 0,C 180,E1 -8352.854,E2 -8352.854} C_VEL
LIN {X 0,Y 452.721,Z 317.643,A -85,B 0,C 180,E1 -8356.078,E2 -8356.078} C_VEL
LIN {X 0,Y 452.668,Z 321.133,A -85,B 0,C 180,E1 -8357.362,E2 -8357.362} C_VEL
LIN {X 0,Y 454.074,Z 333.116,A -85,B 0,C 180,E1 -8357.814,E2 -8357.814} C_VEL
LIN {X 0,Y 454.662,Z 342.4,A -85,B 0,C 180,E1 -8358.284,E2 -8358.284} C_VEL
LIN {X 0,Y 454.347,Z 351.422,A -85,B 0,C 180,E1 -8358.853,E2 -8358.853} C_VEL
LIN {X 0,Y 453.949,Z 359.832,A -85,B 0,C 180,E1 -8359.52,E2 -8359.52} C_VEL
LIN {X 0,Y 453.568,Z 367.784,A -85,B 0,C 180,E1 -8360.3,E2 -8360.3} C_VEL
LIN {X 0,Y 453.276,Z 374.367,A -85,B 0,C 180,E1 -8361.082,E2 -8361.082} C_VEL
LIN {X 0,Y 453.005,Z 380.635,A -85,B 0,C 180,E1 -8361.975,E2 -8361.975} C_VEL
LIN {X 0,Y 452.802,Z 385.848,A -85,B 0,C 180,E1 -8362.868,E2 -8362.868} C_VEL
LIN {X 0,Y 452.653,Z 390.199,A -85,B 0,C 180,E1 -8363.762,E2 -8363.762} C_VEL
LIN {X 0,Y 452.581,Z 395.355,A -85,B 0,C 180,E1 -8365.102,E2 -8365.102} C_VEL
LIN {X 0,Y 452.545,Z 399.138,A -85,B 0,C 180,E1 -8366.44,E2 -8366.44} C_VEL
LIN {X 0,Y 452.534,Z 400.862,A -85,B 0,C 180,E1 -8367.331,E2 -8367.331} C_VEL
LIN {X 0,Y 452.483,Z 402.089,A -85,B 0,C 180,E1 -8368.221,E2 -8368.221} C_VEL
LIN {X 0,Y 452.488,Z 402.844,A -85,B 0,C 180,E1 -8369.111,E2 -8369.111} C_VEL
LIN {X 0,Y 452.467,Z 403.125,A -85,B 0,C 180,E1 -8370.001,E2 -8370.001} C_VEL
LIN {X 0,Y 452.488,Z 402.819,A -85,B 0,C 180,E1 -8370.891,E2 -8370.891} C_VEL
LIN {X 0,Y 452.484,Z 402.001,A -85,B 0,C 180,E1 -8371.781,E2 -8371.781} C_VEL
LIN {X 0,Y 452.534,Z 400.707,A -85,B 0,C 180,E1 -8372.672,E2 -8372.672} C_VEL
LIN {X 0,Y 452.508,Z 397.744,A -85,B 0,C 180,E1 -8374.009,E2 -8374.009} C_VEL
LIN {X 0,Y 452.628,Z 393.508,A -85,B 0,C 180,E1 -8375.347,E2 -8375.347} C_VEL
LIN {X 0,Y 452.764,Z 387.662,A -85,B 0,C 180,E1 -8376.686,E2 -8376.686} C_VEL
LIN {X 0,Y 452.936,Z 381.355,A -85,B 0,C 180,E1 -8377.804,E2 -8377.804} C_VEL
LIN {X 0,Y 453.191,Z 375.191,A -85,B 0,C 180,E1 -8378.698,E2 -8378.698} C_VEL
LIN {X 0,Y 453.43,Z 368.715,A -85,B 0,C 180,E1 -8379.48,E2 -8379.48} C_VEL
LIN {X 0,Y 453.773,Z 360.877,A -85,B 0,C 180,E1 -8380.261,E2 -8380.261} C_VEL
LIN {X 0,Y 454.049,Z 354.12,A -85,B 0,C 180,E1 -8380.818,E2 -8380.818} C_VEL
LIN {X 0,Y 454.329,Z 345.867,A -85,B 0,C 180,E1 -8381.376,E2 -8381.376} C_VEL
LIN {X 0,Y 454.364,Z 338.721,A -85,B 0,C 180,E1 -8381.77,E2 -8381.77} C_VEL
LIN {X 0,Y 453.425,Z 328.816,A -85,B 0,C 180,E1 -8382.203,E2 -8382.203} C_VEL
LIN {X 0,Y 452.661,Z 321.332,A -85,B 0,C 180,E1 -8382.465,E2 -8382.465} C_VEL
LIN {X 0,Y 452.847,Z 312.24,A -85,B 0,C 180,E1 -8385.799,E2 -8385.799} C_VEL
LIN {X 0,Y 453.019,Z 303.567,A -85,B 0,C 180,E1 -8389.014,E2 -8389.014} C_VEL
LIN {X 0,Y 453.337,Z 294.791,A -85,B 0,C 180,E1 -8392.324,E2 -8392.324} C_VEL
LIN {X 0,Y 453.704,Z 286.012,A -85,B 0,C 180,E1 -8395.705,E2 -8395.705} C_VEL
LIN {X 0,Y 454.068,Z 278.513,A -85,B 0,C 180,E1 -8398.674,E2 -8398.674} C_VEL
LIN {X 0,Y 454.51,Z 270.975,A -85,B 0,C 180,E1 -8401.738,E2 -8401.738} C_VEL
LIN {X 0,Y 454.551,Z 267.059,A -85,B 0,C 180,E1 -8403.392,E2 -8403.392} C_VEL
LIN {X 0,Y 453.48,Z 260.813,A -85,B 0,C 180,E1 -8406.221,E2 -8406.221} C_VEL
LIN {X 0,Y 453.491,Z 260.81,A -85,B 0,C 180,E1 -8409.451,E2 -8409.451} C_VEL
LIN {X 0,Y 453.485,Z 260.812,A -85,B 0,C 180,E1 -8411.935,E2 -8411.935} C_VEL
LIN {X 0,Y 453.492,Z 260.81,A -85,B 0,C 180,E1 -8415.471,E2 -8415.471} C_VEL
LIN {X 0,Y 453.488,Z 260.812,A -85,B 0,C 180,E1 -8418.209,E2 -8418.209} C_VEL
LIN {X 0,Y 453.479,Z 260.81,A -85,B 0,C 180,E1 -8420.797,E2 -8420.797} C_VEL
LIN {X 0,Y 453.46,Z 260.815,A -85,B 0,C 180,E1 -8423.917,E2 -8423.917} C_VEL
LIN {X 0,Y 453.49,Z 260.81,A -85,B 0,C 180,E1 -8427.151,E2 -8427.151} C_VEL
LIN {X 0,Y 453.483,Z 260.811,A -85,B 0,C 180,E1 -8430.268,E2 -8430.268} C_VEL
LIN {X 0,Y 453.511,Z 260.809,A -85,B 0,C 180,E1 -8433.293,E2 -8433.293} C_VEL
LIN {X 0,Y 453.506,Z 260.807,A -85,B 0,C 180,E1 -8436.238,E2 -8436.238} C_VEL
LIN {X 0,Y 453.491,Z 260.811,A -85,B 0,C 180,E1 -8439.117,E2 -8439.117} C_VEL
LIN {X 0,Y 453.512,Z 260.806,A -85,B 0,C 180,E1 -8441.943,E2 -8441.943} C_VEL
LIN {X 0,Y 453.547,Z 260.804,A -85,B 0,C 180,E1 -8444.725,E2 -8444.725} C_VEL
LIN {X 0,Y 453.566,Z 260.8,A -85,B 0,C 180,E1 -8448.378,E2 -8448.378} C_VEL
LIN {X 0,Y 453.592,Z 260.798,A -85,B 0,C 180,E1 -8451.085,E2 -8451.085} C_VEL
LIN {X 0,Y 453.672,Z 260.787,A -85,B 0,C 180,E1 -8453.773,E2 -8453.773} C_VEL
LIN {X 0,Y 453.75,Z 260.777,A -85,B 0,C 180,E1 -8457.335,E2 -8457.335} C_VEL
LIN {X 0,Y 453.828,Z 260.768,A -85,B 0,C 180,E1 -8459.998,E2 -8459.998} C_VEL
LIN {X 0,Y 453.77,Z 260.777,A -85,B 0,C 180,E1 -8462.662,E2 -8462.662} C_VEL
LIN {X 0,Y 453.682,Z 260.788,A -85,B 0,C 180,E1 -8466.223,E2 -8466.223} C_VEL
LIN {X 0,Y 453.596,Z 260.797,A -85,B 0,C 180,E1 -8468.911,E2 -8468.911} C_VEL
LIN {X 0,Y 453.566,Z 260.801,A -85,B 0,C 180,E1 -8472.527,E2 -8472.527} C_VEL
LIN {X 0,Y 453.547,Z 260.805,A -85,B 0,C 180,E1 -8476.194,E2 -8476.194} C_VEL
LIN {X 0,Y 453.521,Z 260.805,A -85,B 0,C 180,E1 -8479.038,E2 -8479.038} C_VEL
LIN {X 0,Y 453.476,Z 260.813,A -85,B 0,C 180,E1 -8481.834,E2 -8481.834} C_VEL
LIN {X 0,Y 453.513,Z 260.806,A -85,B 0,C 180,E1 -8484.732,E2 -8484.732} C_VEL
LIN {X 0,Y 453.535,Z 260.806,A -85,B 0,C 180,E1 -8487.959,E2 -8487.959} C_VEL
LIN {X 0,Y 453.463,Z 260.815,A -85,B 0,C 180,E1 -8491.523,E2 -8491.523} C_VEL
LIN {X 0,Y 453.484,Z 260.81,A -85,B 0,C 180,E1 -8494.775,E2 -8494.775} C_VEL
LIN {X 0,Y 453.477,Z 260.811,A -85,B 0,C 180,E1 -8498.307,E2 -8498.307} C_VEL
LIN {X 0,Y 453.509,Z 260.807,A -85,B 0,C 180,E1 -8500.604,E2 -8500.604} C_VEL
LIN {X 0,Y 453.474,Z 260.814,A -85,B 0,C 180,E1 -8503.245,E2 -8503.245} C_VEL
LIN {X 0,Y 453.468,Z 260.813,A -85,B 0,C 180,E1 -8505.778,E2 -8505.778} C_VEL
LIN {X 0,Y 453.487,Z 260.809,A -85,B 0,C 180,E1 -8508.209,E2 -8508.209} C_VEL
LIN {X 0,Y 453.522,Z 260.808,A -85,B 0,C 180,E1 -8510.785,E2 -8510.785} C_VEL
LIN {X 0,Y 453.446,Z 260.814,A -85,B 0,C 180,E1 -8513.915,E2 -8513.915} C_VEL
LIN {X 0,Y 453.47,Z 260.814,A -85,B 0,C 180,E1 -8517.149,E2 -8517.149} C_VEL
LIN {X 0,Y 453.5,Z 260.809,A -85,B 0,C 180,E1 -8520.269,E2 -8520.269} C_VEL
LIN {X 0,Y 453.499,Z 260.81,A -85,B 0,C 180,E1 -8523.292,E2 -8523.292} C_VEL
LIN {X 0,Y 453.492,Z 260.81,A -85,B 0,C 180,E1 -8526.237,E2 -8526.237} C_VEL
LIN {X 0,Y 453.499,Z 260.809,A -85,B 0,C 180,E1 -8529.117,E2 -8529.117} C_VEL
LIN {X 0,Y 453.359,Z 260.827,A -85,B 0,C 180,E1 -8531.937,E2 -8531.937} C_VEL
LIN {X 0,Y 453.031,Z 260.928,A -85,B 0,C 180,E1 -8534.708,E2 -8534.708} C_VEL
LIN {X 0,Y 453.094,Z 264.703,A -85,B 0,C 180,E1 -8537.729,E2 -8537.729} C_VEL
LIN {X 0,Y 452.925,Z 268.95,A -85,B 0,C 180,E1 -8541.072,E2 -8541.072} C_VEL
LIN {X 0,Y 452.946,Z 271.343,A -85,B 0,C 180,E1 -8542.928,E2 -8542.928} C_VEL
LIN {X 0,Y 452.31,Z 272.341,A -85,B 0,C 180,E1 -8543.66,E2 -8543.66} C_VEL
LIN {X 0,Y 449.445,Z 274.12,A -85,B 0,C 180,E1 -8544.844,E2 -8544.844} C_VEL
LIN {X 0,Y 446.969,Z 275.561,A -85,B 0,C 180,E1 -8545.799,E2 -8545.799} C_VEL
LIN {X 0,Y 445.862,Z 276.608,A -85,B 0,C 180,E1 -8546.539,E2 -8546.539} C_VEL
LIN {X 0,Y 445.749,Z 276.943,A -85,B 0,C 180,E1 -8546.79,E2 -8546.79} C_VEL
LIN {X 0,Y 445.491,Z 281.182,A -85,B 0,C 180,E1 -8549.999,E2 -8549.999} C_VEL
LIN {X 0,Y 445.492,Z 283.163,A -85,B 0,C 180,E1 -8551.496,E2 -8551.496} C_VEL
LIN {X 0,Y 447.634,Z 295.229,A -85,B 0,C 180,E1 -8552.023,E2 -8552.023} C_VEL
LIN {X 0,Y 447.771,Z 299.833,A -85,B 0,C 180,E1 -8552.248,E2 -8552.248} C_VEL
LIN {X 0,Y 447.475,Z 310.515,A -85,B 0,C 180,E1 -8552.925,E2 -8552.925} C_VEL
LIN {X 0,Y 447.121,Z 318.883,A -85,B 0,C 180,E1 -8553.604,E2 -8553.604} C_VEL
LIN {X 0,Y 446.756,Z 326.794,A -85,B 0,C 180,E1 -8554.397,E2 -8554.397} C_VEL
LIN {X 0,Y 446.557,Z 333.295,A -85,B 0,C 180,E1 -8555.191,E2 -8555.191} C_VEL
LIN {X 0,Y 446.249,Z 339.509,A -85,B 0,C 180,E1 -8556.101,E2 -8556.101} C_VEL
LIN {X 0,Y 446.087,Z 344.701,A -85,B 0,C 180,E1 -8557.021,E2 -8557.021} C_VEL
LIN {X 0,Y 445.954,Z 347.988,A -85,B 0,C 180,E1 -8557.697,E2 -8557.697} C_VEL
LIN {X 0,Y 445.742,Z 351.757,A -85,B 0,C 180,E1 -8558.613,E2 -8558.613} C_VEL
LIN {X 0,Y 445.56,Z 356.025,A -85,B 0,C 180,E1 -8559.991,E2 -8559.991} C_VEL
LIN {X 0,Y 445.507,Z 358.186,A -85,B 0,C 180,E1 -8560.911,E2 -8560.911} C_VEL
LIN {X 0,Y 445.454,Z 360,A -85,B 0,C 180,E1 -8562.004,E2 -8562.004} C_VEL
LIN {X 0,Y 445.359,Z 360.812,A -85,B 0,C 180,E1 -8562.762,E2 -8562.762} C_VEL
LIN {X 0,Y 445.354,Z 361.292,A -85,B 0,C 180,E1 -8563.691,E2 -8563.691} C_VEL
LIN {X 0,Y 445.359,Z 361.282,A -85,B 0,C 180,E1 -8564.623,E2 -8564.623} C_VEL
LIN {X 0,Y 445.408,Z 360.575,A -85,B 0,C 180,E1 -8565.75,E2 -8565.75} C_VEL
LIN {X 0,Y 445.479,Z 359.747,A -85,B 0,C 180,E1 -8566.496,E2 -8566.496} C_VEL
LIN {X 0,Y 445.621,Z 357.021,A -85,B 0,C 180,E1 -8567.91,E2 -8567.91} C_VEL
LIN {X 0,Y 445.827,Z 352.94,A -85,B 0,C 180,E1 -8569.331,E2 -8569.331} C_VEL
LIN {X 0,Y 446.03,Z 348.35,A -85,B 0,C 180,E1 -8570.522,E2 -8570.522} C_VEL
LIN {X 0,Y 446.395,Z 341.383,A -85,B 0,C 180,E1 -8571.904,E2 -8571.904} C_VEL
LIN {X 0,Y 446.71,Z 334.826,A -85,B 0,C 180,E1 -8572.915,E2 -8572.915} C_VEL
LIN {X 0,Y 447.078,Z 327.142,A -85,B 0,C 180,E1 -8573.876,E2 -8573.876} C_VEL
LIN {X 0,Y 447.432,Z 319.666,A -85,B 0,C 180,E1 -8574.64,E2 -8574.64} C_VEL
LIN {X 0,Y 447.842,Z 311.527,A -85,B 0,C 180,E1 -8575.316,E2 -8575.316} C_VEL
LIN {X 0,Y 448.189,Z 302.425,A -85,B 0,C 180,E1 -8575.918,E2 -8575.918} C_VEL
LIN {X 0,Y 448.247,Z 297.646,A -85,B 0,C 180,E1 -8576.176,E2 -8576.176} C_VEL
LIN {X 0,Y 446.609,Z 288.526,A -85,B 0,C 180,E1 -8576.63,E2 -8576.63} C_VEL
LIN {X 0,Y 445.535,Z 283.391,A -85,B 0,C 180,E1 -8576.857,E2 -8576.857} C_VEL
LIN {X 0,Y 445.608,Z 278.965,A -85,B 0,C 180,E1 -8580.309,E2 -8580.309} C_VEL
LIN {X 0,Y 445.66,Z 274.962,A -85,B 0,C 180,E1 -8583.499,E2 -8583.499} C_VEL
LIN {X 0,Y 445.765,Z 270.914,A -85,B 0,C 180,E1 -8586.805,E2 -8586.805} C_VEL
LIN {X 0,Y 445.88,Z 266.754,A -85,B 0,C 180,E1 -8590.257,E2 -8590.257} C_VEL
LIN {X 0,Y 446.031,Z 262.879,A -85,B 0,C 180,E1 -8593.55,E2 -8593.55} C_VEL
LIN {X 0,Y 446.106,Z 261.731,A -85,B 0,C 180,E1 -8594.855,E2 -8594.855} C_VEL
LIN {X 0,Y 446.356,Z 261.699,A -85,B 0,C 180,E1 -8597.731,E2 -8597.731} C_VEL
LIN {X 0,Y 446.455,Z 261.688,A -85,B 0,C 180,E1 -8600.977,E2 -8600.977} C_VEL
LIN {X 0,Y 446.402,Z 261.695,A -85,B 0,C 180,E1 -8604.375,E2 -8604.375} C_VEL
LIN {X 0,Y 446.403,Z 261.694,A -85,B 0,C 180,E1 -8607.64,E2 -8607.64} C_VEL
LIN {X 0,Y 446.43,Z 261.689,A -85,B 0,C 180,E1 -8610.792,E2 -8610.792} C_VEL
LIN {X 0,Y 446.46,Z 261.687,A -85,B 0,C 180,E1 -8613.85,E2 -8613.85} C_VEL
LIN {X 0,Y 446.411,Z 261.691,A -85,B 0,C 180,E1 -8616.825,E2 -8616.825} C_VEL
LIN {X 0,Y 446.428,Z 261.687,A -85,B 0,C 180,E1 -8619.739,E2 -8619.739} C_VEL
LIN {X 0,Y 446.448,Z 261.683,A -85,B 0,C 180,E1 -8622.599,E2 -8622.599} C_VEL
LIN {X 0,Y 446.454,Z 261.682,A -85,B 0,C 180,E1 -8625.414,E2 -8625.414} C_VEL
LIN {X 0,Y 446.526,Z 261.677,A -85,B 0,C 180,E1 -8628.195,E2 -8628.195} C_VEL
LIN {X 0,Y 446.562,Z 261.671,A -85,B 0,C 180,E1 -8631.859,E2 -8631.859} C_VEL
LIN {X 0,Y 446.622,Z 261.666,A -85,B 0,C 180,E1 -8634.584,E2 -8634.584} C_VEL
LIN {X 0,Y 446.7,Z 261.655,A -85,B 0,C 180,E1 -8637.296,E2 -8637.296} C_VEL
LIN {X 0,Y 446.781,Z 261.644,A -85,B 0,C 180,E1 -8640.002,E2 -8640.002} C_VEL
LIN {X 0,Y 446.679,Z 261.656,A -85,B 0,C 180,E1 -8642.707,E2 -8642.707} C_VEL
LIN {X 0,Y 446.637,Z 261.658,A -85,B 0,C 180,E1 -8646.325,E2 -8646.325} C_VEL
LIN {X 0,Y 446.526,Z 261.676,A -85,B 0,C 180,E1 -8649.057,E2 -8649.057} C_VEL
LIN {X 0,Y 446.525,Z 261.676,A -85,B 0,C 180,E1 -8652.731,E2 -8652.731} C_VEL
LIN {X 0,Y 446.48,Z 261.685,A -85,B 0,C 180,E1 -8656.461,E2 -8656.461} C_VEL
LIN {X 0,Y 446.459,Z 261.685,A -85,B 0,C 180,E1 -8659.305,E2 -8659.305} C_VEL
LIN {X 0,Y 446.41,Z 261.69,A -85,B 0,C 180,E1 -8662.201,E2 -8662.201} C_VEL
LIN {X 0,Y 446.438,Z 261.687,A -85,B 0,C 180,E1 -8665.155,E2 -8665.155} C_VEL
LIN {X 0,Y 446.441,Z 261.688,A -85,B 0,C 180,E1 -8668.183,E2 -8668.183} C_VEL
LIN {X 0,Y 446.41,Z 261.693,A -85,B 0,C 180,E1 -8671.302,E2 -8671.302} C_VEL
LIN {X 0,Y 446.422,Z 261.692,A -85,B 0,C 180,E1 -8674.525,E2 -8674.525} C_VEL
LIN {X 0,Y 446.415,Z 261.691,A -85,B 0,C 180,E1 -8678.082,E2 -8678.082} C_VEL
LIN {X 0,Y 446.439,Z 261.687,A -85,B 0,C 180,E1 -8680.922,E2 -8680.922} C_VEL
LIN {X 0,Y 446.395,Z 261.696,A -85,B 0,C 180,E1 -8683.848,E2 -8683.848} C_VEL
LIN {X 0,Y 446.394,Z 261.693,A -85,B 0,C 180,E1 -8686.405,E2 -8686.405} C_VEL
LIN {X 0,Y 446.424,Z 261.691,A -85,B 0,C 180,E1 -8689.084,E2 -8689.084} C_VEL
LIN {X 0,Y 446.406,Z 261.695,A -85,B 0,C 180,E1 -8692.123,E2 -8692.123} C_VEL
LIN {X 0,Y 446.436,Z 261.836,A -85,B 0,C 180,E1 -8692.411,E2 -8692.411} C_VEL
LIN {X 0,Y 447.581,Z 268.054,A -85,B 0,C 180,E1 -8695.58,E2 -8695.58} C_VEL
LIN {X 0,Y 447.894,Z 271.547,A -85,B 0,C 180,E1 -8697.226,E2 -8697.226} C_VEL
LIN {X 0,Y 447.466,Z 277.382,A -85,B 0,C 180,E1 -8699.83,E2 -8699.83} C_VEL
LIN {X 0,Y 446.962,Z 284.523,A -85,B 0,C 180,E1 -8702.873,E2 -8702.873} C_VEL
LIN {X 0,Y 446.51,Z 293.003,A -85,B 0,C 180,E1 -8706.363,E2 -8706.363} C_VEL
LIN {X 0,Y 446.11,Z 301.468,A -85,B 0,C 180,E1 -8709.723,E2 -8709.723} C_VEL
LIN {X 0,Y 445.854,Z 310.04,A -85,B 0,C 180,E1 -8713.047,E2 -8713.047} C_VEL
LIN {X 0,Y 445.618,Z 318.645,A -85,B 0,C 180,E1 -8716.317,E2 -8716.317} C_VEL
LIN {X 0,Y 445.586,Z 320.79,A -85,B 0,C 180,E1 -8717.129,E2 -8717.129} C_VEL
LIN {X 0,Y 447.081,Z 332.789,A -85,B 0,C 180,E1 -8717.592,E2 -8717.592} C_VEL
LIN {X 0,Y 447.7,Z 342.679,A -85,B 0,C 180,E1 -8718.11,E2 -8718.11} C_VEL
LIN {X 0,Y 447.389,Z 351.418,A -85,B 0,C 180,E1 -8718.677,E2 -8718.677} C_VEL
LIN {X 0,Y 446.969,Z 359.759,A -85,B 0,C 180,E1 -8719.355,E2 -8719.355} C_VEL
LIN {X 0,Y 446.571,Z 367.659,A -85,B 0,C 180,E1 -8720.147,E2 -8720.147} C_VEL
LIN {X 0,Y 446.263,Z 374.2,A -85,B 0,C 180,E1 -8720.94,E2 -8720.94} C_VEL
LIN {X 0,Y 445.951,Z 380.439,A -85,B 0,C 180,E1 -8721.847,E2 -8721.847} C_VEL
LIN {X 0,Y 445.757,Z 385.629,A -85,B 0,C 180,E1 -8722.755,E2 -8722.755} C_VEL
LIN {X 0,Y 445.579,Z 389.959,A -85,B 0,C 180,E1 -8723.662,E2 -8723.662} C_VEL
LIN {X 0,Y 445.513,Z 395.097,A -85,B 0,C 180,E1 -8725.024,E2 -8725.024} C_VEL
LIN {X 0,Y 445.439,Z 398.859,A -85,B 0,C 180,E1 -8726.383,E2 -8726.383} C_VEL
LIN {X 0,Y 445.459,Z 400.571,A -85,B 0,C 180,E1 -8727.288,E2 -8727.288} C_VEL
LIN {X 0,Y 445.4,Z 401.782,A -85,B 0,C 180,E1 -8728.193,E2 -8728.193} C_VEL
LIN {X 0,Y 445.395,Z 402.521,A -85,B 0,C 180,E1 -8729.097,E2 -8729.097} C_VEL
LIN {X 0,Y 445.403,Z 402.792,A -85,B 0,C 180,E1 -8730.001,E2 -8730.001} C_VEL
LIN {X 0,Y 445.395,Z 402.482,A -85,B 0,C 180,E1 -8730.905,E2 -8730.905} C_VEL
LIN {X 0,Y 445.4,Z 401.648,A -85,B 0,C 180,E1 -8731.81,E2 -8731.81} C_VEL
LIN {X 0,Y 445.46,Z 400.338,A -85,B 0,C 180,E1 -8732.714,E2 -8732.714} C_VEL
LIN {X 0,Y 445.414,Z 397.357,A -85,B 0,C 180,E1 -8734.073,E2 -8734.073} C_VEL
LIN {X 0,Y 445.542,Z 393.103,A -85,B 0,C 180,E1 -8735.432,E2 -8735.432} C_VEL
LIN {X 0,Y 445.707,Z 387.216,A -85,B 0,C 180,E1 -8736.792,E2 -8736.792} C_VEL
LIN {X 0,Y 445.878,Z 380.884,A -85,B 0,C 180,E1 -8737.929,E2 -8737.929} C_VEL
LIN {X 0,Y 446.141,Z 374.691,A -85,B 0,C 180,E1 -8738.836,E2 -8738.836} C_VEL
LIN {X 0,Y 446.391,Z 368.18,A -85,B 0,C 180,E1 -8739.631,E2 -8739.631} C_VEL
LIN {X 0,Y 446.719,Z 360.297,A -85,B 0,C 180,E1 -8740.425,E2 -8740.425} C_VEL
LIN {X 0,Y 447.132,Z 351.985,A -85,B 0,C 180,E1 -8741.102,E2 -8741.102} C_VEL
LIN {X 0,Y 447.473,Z 341.387,A -85,B 0,C 180,E1 -8741.782,E2 -8741.782} C_VEL
LIN {X 0,Y 446.496,Z 330.181,A -85,B 0,C 180,E1 -8742.312,E2 -8742.312} C_VEL
LIN {X 0,Y 445.573,Z 321.075,A -85,B 0,C 180,E1 -8742.62,E2 -8742.62} C_VEL
LIN {X 0,Y 445.756,Z 312.303,A -85,B 0,C 180,E1 -8745.896,E2 -8745.896} C_VEL
LIN {X 0,Y 445.984,Z 303.244,A -85,B 0,C 180,E1 -8749.326,E2 -8749.326} C_VEL
LIN {X 0,Y 446.308,Z 294.46,A -85,B 0,C 180,E1 -8752.694,E2 -8752.694} C_VEL
LIN {X 0,Y 446.724,Z 285.41,A -85,B 0,C 180,E1 -8756.266,E2 -8756.266} C_VEL
LIN {X 0,Y 447.204,Z 276.978,A -85,B 0,C 180,E1 -8759.673,E2 -8759.673} C_VEL
LIN {X 0,Y 447.545,Z 270.772,A -85,B 0,C 180,E1 -8762.272,E2 -8762.272} C_VEL
LIN {X 0,Y 447.455,Z 267.587,A -85,B 0,C 180,E1 -8763.648,E2 -8763.648} C_VEL
LIN {X 0,Y 446.418,Z 261.693,A -85,B 0,C 180,E1 -8766.348,E2 -8766.348} C_VEL
LIN {X 0,Y 446.458,Z 261.687,A -85,B 0,C 180,E1 -8769.524,E2 -8769.524} C_VEL
LIN {X 0,Y 446.437,Z 261.688,A -85,B 0,C 180,E1 -8772.605,E2 -8772.605} C_VEL
LIN {X 0,Y 446.459,Z 261.684,A -85,B 0,C 180,E1 -8775.104,E2 -8775.104} C_VEL
LIN {X 0,Y 446.437,Z 261.687,A -85,B 0,C 180,E1 -8778.609,E2 -8778.609} C_VEL
LIN {X 0,Y 446.434,Z 261.688,A -85,B 0,C 180,E1 -8780.971,E2 -8780.971} C_VEL
LIN {X 0,Y 446.426,Z 261.69,A -85,B 0,C 180,E1 -8784.373,E2 -8784.373} C_VEL
LIN {X 0,Y 446.43,Z 261.691,A -85,B 0,C 180,E1 -8787.638,E2 -8787.638} C_VEL
LIN {X 0,Y 446.457,Z 261.686,A -85,B 0,C 180,E1 -8790.79,E2 -8790.79} C_VEL
LIN {X 0,Y 446.487,Z 261.682,A -85,B 0,C 180,E1 -8793.848,E2 -8793.848} C_VEL
LIN {X 0,Y 446.435,Z 261.689,A -85,B 0,C 180,E1 -8796.822,E2 -8796.822} C_VEL
LIN {X 0,Y 446.452,Z 261.686,A -85,B 0,C 180,E1 -8799.736,E2 -8799.736} C_VEL
LIN {X 0,Y 446.465,Z 261.685,A -85,B 0,C 180,E1 -8802.596,E2 -8802.596} C_VEL
LIN {X 0,Y 446.477,Z 261.685,A -85,B 0,C 180,E1 -8805.411,E2 -8805.411} C_VEL
LIN {X 0,Y 446.525,Z 261.677,A -85,B 0,C 180,E1 -8808.192,E2 -8808.192} C_VEL
LIN {X 0,Y 446.539,Z 261.678,A -85,B 0,C 180,E1 -8810.943,E2 -8810.943} C_VEL
LIN {X 0,Y 446.641,Z 261.662,A -85,B 0,C 180,E1 -8813.675,E2 -8813.675} C_VEL
LIN {X 0,Y 446.697,Z 261.656,A -85,B 0,C 180,E1 -8817.293,E2 -8817.293} C_VEL
LIN {X 0,Y 446.798,Z 261.643,A -85,B 0,C 180,E1 -8819.998,E2 -8819.998} C_VEL
LIN {X 0,Y 446.714,Z 261.656,A -85,B 0,C 180,E1 -8822.704,E2 -8822.704} C_VEL
LIN {X 0,Y 446.651,Z 261.663,A -85,B 0,C 180,E1 -8826.322,E2 -8826.322} C_VEL
LIN {X 0,Y 446.542,Z 261.675,A -85,B 0,C 180,E1 -8829.053,E2 -8829.053} C_VEL
LIN {X 0,Y 446.524,Z 261.679,A -85,B 0,C 180,E1 -8832.728,E2 -8832.728} C_VEL
LIN {X 0,Y 446.498,Z 261.683,A -85,B 0,C 180,E1 -8836.226,E2 -8836.226} C_VEL
LIN {X 0,Y 446.47,Z 261.684,A -85,B 0,C 180,E1 -8839.301,E2 -8839.301} C_VEL
LIN {X 0,Y 446.418,Z 261.692,A -85,B 0,C 180,E1 -8842.197,E2 -8842.197} C_VEL
LIN {X 0,Y 446.456,Z 261.685,A -85,B 0,C 180,E1 -8845.15,E2 -8845.15} C_VEL
LIN {X 0,Y 446.482,Z 261.684,A -85,B 0,C 180,E1 -8848.176,E2 -8848.176} C_VEL
LIN {X 0,Y 446.416,Z 261.692,A -85,B 0,C 180,E1 -8851.773,E2 -8851.773} C_VEL
LIN {X 0,Y 446.426,Z 261.689,A -85,B 0,C 180,E1 -8854.521,E2 -8854.521} C_VEL
LIN {X 0,Y 446.431,Z 261.69,A -85,B 0,C 180,E1 -8858.08,E2 -8858.08} C_VEL
LIN {X 0,Y 446.44,Z 261.689,A -85,B 0,C 180,E1 -8860.918,E2 -8860.918} C_VEL
LIN {X 0,Y 446.437,Z 261.689,A -85,B 0,C 180,E1 -8863.838,E2 -8863.838} C_VEL
LIN {X 0,Y 446.438,Z 261.688,A -85,B 0,C 180,E1 -8866.395,E2 -8866.395} C_VEL
LIN {X 0,Y 446.459,Z 261.685,A -85,B 0,C 180,E1 -8869.803,E2 -8869.803} C_VEL
LIN {X 0,Y 446.424,Z 261.688,A -85,B 0,C 180,E1 -8872.122,E2 -8872.122} C_VEL
LIN {X 0,Y 446.418,Z 261.691,A -85,B 0,C 180,E1 -8875.475,E2 -8875.475} C_VEL
LIN {X 0,Y 446.407,Z 261.695,A -85,B 0,C 180,E1 -8878.698,E2 -8878.698} C_VEL
LIN {X 0,Y 446.47,Z 261.683,A -85,B 0,C 180,E1 -8881.819,E2 -8881.819} C_VEL
LIN {X 0,Y 446.445,Z 261.689,A -85,B 0,C 180,E1 -8884.846,E2 -8884.846} C_VEL
LIN {X 0,Y 446.469,Z 261.685,A -85,B 0,C 180,E1 -8888.231,E2 -8888.231} C_VEL
LIN {X 0,Y 446.441,Z 261.689,A -85,B 0,C 180,E1 -8890.82,E2 -8890.82} C_VEL
LIN {X 0,Y 446.11,Z 261.731,A -85,B 0,C 180,E1 -8893.934,E2 -8893.934} C_VEL
LIN {X 0,Y 446.035,Z 261.741,A -85,B 0,C 180,E1 -8894.462,E2 -8894.462} C_VEL
LIN {X 0,Y 445.925,Z 262.492,A -85,B 0,C 180,E1 -8895.393,E2 -8895.393} C_VEL
LIN {X 0,Y 445.964,Z 265.935,A -85,B 0,C 180,E1 -8898.177,E2 -8898.177} C_VEL
LIN {X 0,Y 445.86,Z 270.584,A -85,B 0,C 180,E1 -8901.843,E2 -8901.843} C_VEL
LIN {X 0,Y 445.895,Z 272.902,A -85,B 0,C 180,E1 -8903.664,E2 -8903.664} C_VEL
LIN {X 0,Y 445.813,Z 276.411,A -85,B 0,C 180,E1 -8906.384,E2 -8906.384} C_VEL
LIN {X 0,Y 445.749,Z 276.943,A -85,B 0,C 180,E1 -8906.79,E2 -8906.79} C_VEL
LIN {X 0,Y 444.994,Z 277.973,A -85,B 0,C 180,E1 -8907.532,E2 -8907.532} C_VEL
LIN {X 0,Y 442.007,Z 279.785,A -85,B 0,C 180,E1 -8908.731,E2 -8908.731} C_VEL
LIN {X 0,Y 439.531,Z 281.244,A -85,B 0,C 180,E1 -8909.698,E2 -8909.698} C_VEL
LIN {X 0,Y 438.49,Z 282.304,A -85,B 0,C 180,E1 -8910.448,E2 -8910.448} C_VEL
LIN {X 0,Y 438.416,Z 282.644,A -85,B 0,C 180,E1 -8910.703,E2 -8910.703} C_VEL
LIN {X 0,Y 438.418,Z 283.453,A -85,B 0,C 180,E1 -8911.319,E2 -8911.319} C_VEL
LIN {X 0,Y 440.468,Z 294.97,A -85,B 0,C 180,E1 -8911.827,E2 -8911.827} C_VEL
LIN {X 0,Y 440.818,Z 299.485,A -85,B 0,C 180,E1 -8912.055,E2 -8912.055} C_VEL
LIN {X 0,Y 440.501,Z 310.394,A -85,B 0,C 180,E1 -8912.742,E2 -8912.742} C_VEL
LIN {X 0,Y 440.156,Z 318.833,A -85,B 0,C 180,E1 -8913.431,E2 -8913.431} C_VEL
LIN {X 0,Y 439.747,Z 326.815,A -85,B 0,C 180,E1 -8914.238,E2 -8914.238} C_VEL
LIN {X 0,Y 439.548,Z 333.364,A -85,B 0,C 180,E1 -8915.044,E2 -8915.044} C_VEL
LIN {X 0,Y 439.2,Z 339.626,A -85,B 0,C 180,E1 -8915.969,E2 -8915.969} C_VEL
LIN {X 0,Y 439.081,Z 344.408,A -85,B 0,C 180,E1 -8916.817,E2 -8916.817} C_VEL
LIN {X 0,Y 438.844,Z 349.135,A -85,B 0,C 180,E1 -8917.822,E2 -8917.822} C_VEL
LIN {X 0,Y 438.634,Z 352.739,A -85,B 0,C 180,E1 -8918.754,E2 -8918.754} C_VEL
LIN {X 0,Y 438.472,Z 356.85,A -85,B 0,C 180,E1 -8920.154,E2 -8920.154} C_VEL
LIN {X 0,Y 438.397,Z 358.868,A -85,B 0,C 180,E1 -8921.09,E2 -8921.09} C_VEL
LIN {X 0,Y 438.366,Z 360.396,A -85,B 0,C 180,E1 -8922.063,E2 -8922.063} C_VEL
LIN {X 0,Y 438.271,Z 361.33,A -85,B 0,C 180,E1 -8922.972,E2 -8922.972} C_VEL
LIN {X 0,Y 438.276,Z 361.694,A -85,B 0,C 180,E1 -8923.917,E2 -8923.917} C_VEL
LIN {X 0,Y 438.293,Z 361.543,A -85,B 0,C 180,E1 -8924.865,E2 -8924.865} C_VEL
LIN {X 0,Y 438.352,Z 360.847,A -85,B 0,C 180,E1 -8925.863,E2 -8925.863} C_VEL
LIN {X 0,Y 438.42,Z 359.736,A -85,B 0,C 180,E1 -8926.769,E2 -8926.769} C_VEL
LIN {X 0,Y 438.509,Z 358.024,A -85,B 0,C 180,E1 -8927.727,E2 -8927.727} C_VEL
LIN {X 0,Y 438.73,Z 354.468,A -85,B 0,C 180,E1 -8929.079,E2 -8929.079} C_VEL
LIN {X 0,Y 438.92,Z 350.817,A -85,B 0,C 180,E1 -8930.135,E2 -8930.135} C_VEL
LIN {X 0,Y 439.178,Z 345.452,A -85,B 0,C 180,E1 -8931.348,E2 -8931.348} C_VEL
LIN {X 0,Y 439.497,Z 339.813,A -85,B 0,C 180,E1 -8932.372,E2 -8932.372} C_VEL
LIN {X 0,Y 439.828,Z 333.635,A -85,B 0,C 180,E1 -8933.294,E2 -8933.294} C_VEL
LIN {X 0,Y 440.164,Z 326.715,A -85,B 0,C 180,E1 -8934.15,E2 -8934.15} C_VEL
LIN {X 0,Y 440.6,Z 318.776,A -85,B 0,C 180,E1 -8934.953,E2 -8934.953} C_VEL
LIN {X 0,Y 441.033,Z 309.204,A -85,B 0,C 180,E1 -8935.73,E2 -8935.73} C_VEL
LIN {X 0,Y 441.369,Z 299.001,A -85,B 0,C 180,E1 -8936.349,E2 -8936.349} C_VEL
LIN {X 0,Y 439.578,Z 288.939,A -85,B 0,C 180,E1 -8936.865,E2 -8936.865} C_VEL
LIN {X 0,Y 438.456,Z 283.714,A -85,B 0,C 180,E1 -8937.113,E2 -8937.113} C_VEL
LIN {X 0,Y 438.561,Z 279.936,A -85,B 0,C 180,E1 -8940.082,E2 -8940.082} C_VEL
LIN {X 0,Y 438.591,Z 276.286,A -85,B 0,C 180,E1 -8943.01,E2 -8943.01} C_VEL
LIN {X 0,Y 438.695,Z 272.241,A -85,B 0,C 180,E1 -8946.35,E2 -8946.35} C_VEL
LIN {X 0,Y 438.815,Z 268.066,A -85,B 0,C 180,E1 -8949.837,E2 -8949.837} C_VEL
LIN {X 0,Y 438.953,Z 264.884,A -85,B 0,C 180,E1 -8952.57,E2 -8952.57} C_VEL
LIN {X 0,Y 439.058,Z 262.609,A -85,B 0,C 180,E1 -8954.771,E2 -8954.771} C_VEL
LIN {X 0,Y 439.324,Z 262.575,A -85,B 0,C 180,E1 -8957.79,E2 -8957.79} C_VEL
LIN {X 0,Y 439.431,Z 262.56,A -85,B 0,C 180,E1 -8960.231,E2 -8960.231} C_VEL
LIN {X 0,Y 439.358,Z 262.57,A -85,B 0,C 180,E1 -8963.714,E2 -8963.714} C_VEL
LIN {X 0,Y 439.353,Z 262.571,A -85,B 0,C 180,E1 -8967.055,E2 -8967.055} C_VEL
LIN {X 0,Y 439.364,Z 262.569,A -85,B 0,C 180,E1 -8970.275,E2 -8970.275} C_VEL
LIN {X 0,Y 439.411,Z 262.563,A -85,B 0,C 180,E1 -8973.398,E2 -8973.398} C_VEL
LIN {X 0,Y 439.368,Z 262.566,A -85,B 0,C 180,E1 -8976.431,E2 -8976.431} C_VEL
LIN {X 0,Y 439.372,Z 262.565,A -85,B 0,C 180,E1 -8979.399,E2 -8979.399} C_VEL
LIN {X 0,Y 439.416,Z 262.559,A -85,B 0,C 180,E1 -8982.311,E2 -8982.311} C_VEL
LIN {X 0,Y 439.431,Z 262.558,A -85,B 0,C 180,E1 -8985.175,E2 -8985.175} C_VEL
LIN {X 0,Y 439.494,Z 262.556,A -85,B 0,C 180,E1 -8988.004,E2 -8988.004} C_VEL
LIN {X 0,Y 439.52,Z 262.549,A -85,B 0,C 180,E1 -8991.728,E2 -8991.728} C_VEL
LIN {X 0,Y 439.597,Z 262.541,A -85,B 0,C 180,E1 -8994.497,E2 -8994.497} C_VEL
LIN {X 0,Y 439.626,Z 262.532,A -85,B 0,C 180,E1 -8998.169,E2 -8998.169} C_VEL
LIN {X 0,Y 439.751,Z 262.519,A -85,B 0,C 180,E1 -9000.002,E2 -9000.002} C_VEL
LIN {X 0,Y 439.629,Z 262.534,A -85,B 0,C 180,E1 -9002.75,E2 -9002.75} C_VEL
LIN {X 0,Y 439.609,Z 262.534,A -85,B 0,C 180,E1 -9006.427,E2 -9006.427} C_VEL
LIN {X 0,Y 439.489,Z 262.552,A -85,B 0,C 180,E1 -9009.203,E2 -9009.203} C_VEL
LIN {X 0,Y 439.495,Z 262.551,A -85,B 0,C 180,E1 -9012.728,E2 -9012.728} C_VEL
LIN {X 0,Y 439.437,Z 262.561,A -85,B 0,C 180,E1 -9016.35,E2 -9016.35} C_VEL
LIN {X 0,Y 439.393,Z 262.568,A -85,B 0,C 180,E1 -9019.628,E2 -9019.628} C_VEL
LIN {X 0,Y 439.357,Z 262.57,A -85,B 0,C 180,E1 -9022.577,E2 -9022.577} C_VEL
LIN {X 0,Y 439.375,Z 262.568,A -85,B 0,C 180,E1 -9025.588,E2 -9025.588} C_VEL
LIN {X 0,Y 439.393,Z 262.566,A -85,B 0,C 180,E1 -9028.676,E2 -9028.676} C_VEL
LIN {X 0,Y 439.365,Z 262.572,A -85,B 0,C 180,E1 -9032.032,E2 -9032.032} C_VEL
LIN {X 0,Y 439.387,Z 262.571,A -85,B 0,C 180,E1 -9035.342,E2 -9035.342} C_VEL
LIN {X 0,Y 439.386,Z 262.57,A -85,B 0,C 180,E1 -9038.596,E2 -9038.596} C_VEL
LIN {X 0,Y 439.394,Z 262.565,A -85,B 0,C 180,E1 -9041.26,E2 -9041.26} C_VEL
LIN {X 0,Y 439.395,Z 262.57,A -85,B 0,C 180,E1 -9044.731,E2 -9044.731} C_VEL
LIN {X 0,Y 439.392,Z 262.57,A -85,B 0,C 180,E1 -9047.797,E2 -9047.797} C_VEL
LIN {X 0,Y 439.423,Z 262.563,A -85,B 0,C 180,E1 -9050.229,E2 -9050.229} C_VEL
LIN {X 0,Y 439.401,Z 262.764,A -85,B 0,C 180,E1 -9052.138,E2 -9052.138} C_VEL
LIN {X 0,Y 440.597,Z 269.234,A -85,B 0,C 180,E1 -9055.512,E2 -9055.512} C_VEL
LIN {X 0,Y 440.919,Z 272.702,A -85,B 0,C 180,E1 -9057.186,E2 -9057.186} C_VEL
LIN {X 0,Y 440.539,Z 277.748,A -85,B 0,C 180,E1 -9059.483,E2 -9059.483} C_VEL
LIN {X 0,Y 439.993,Z 284.462,A -85,B 0,C 180,E1 -9062.407,E2 -9062.407} C_VEL
LIN {X 0,Y 439.537,Z 292.274,A -85,B 0,C 180,E1 -9065.702,E2 -9065.702} C_VEL
LIN {X 0,Y 439.071,Z 301.31,A -85,B 0,C 180,E1 -9069.383,E2 -9069.383} C_VEL
LIN {X 0,Y 438.779,Z 309.874,A -85,B 0,C 180,E1 -9072.765,E2 -9072.765} C_VEL
LIN {X 0,Y 438.559,Z 318.424,A -85,B 0,C 180,E1 -9076.093,E2 -9076.093} C_VEL
LIN {X 0,Y 438.523,Z 320.497,A -85,B 0,C 180,E1 -9076.888,E2 -9076.888} C_VEL
LIN {X 0,Y 440.129,Z 333.337,A -85,B 0,C 180,E1 -9077.405,E2 -9077.405} C_VEL
LIN {X 0,Y 440.755,Z 342.95,A -85,B 0,C 180,E1 -9077.928,E2 -9077.928} C_VEL
LIN {X 0,Y 440.444,Z 351.475,A -85,B 0,C 180,E1 -9078.496,E2 -9078.496} C_VEL
LIN {X 0,Y 439.996,Z 359.744,A -85,B 0,C 180,E1 -9079.184,E2 -9079.184} C_VEL
LIN {X 0,Y 439.575,Z 367.59,A -85,B 0,C 180,E1 -9079.988,E2 -9079.988} C_VEL
LIN {X 0,Y 439.251,Z 374.087,A -85,B 0,C 180,E1 -9080.794,E2 -9080.794} C_VEL
LIN {X 0,Y 438.913,Z 380.284,A -85,B 0,C 180,E1 -9081.716,E2 -9081.716} C_VEL
LIN {X 0,Y 438.704,Z 385.438,A -85,B 0,C 180,E1 -9082.638,E2 -9082.638} C_VEL
LIN {X 0,Y 438.507,Z 389.738,A -85,B 0,C 180,E1 -9083.56,E2 -9083.56} C_VEL
LIN {X 0,Y 438.464,Z 393.318,A -85,B 0,C 180,E1 -9084.482,E2 -9084.482} C_VEL
LIN {X 0,Y 438.324,Z 397.427,A -85,B 0,C 180,E1 -9085.864,E2 -9085.864} C_VEL
LIN {X 0,Y 438.386,Z 400.283,A -85,B 0,C 180,E1 -9087.245,E2 -9087.245} C_VEL
LIN {X 0,Y 438.32,Z 401.476,A -85,B 0,C 180,E1 -9088.164,E2 -9088.164} C_VEL
LIN {X 0,Y 438.306,Z 402.198,A -85,B 0,C 180,E1 -9089.082,E2 -9089.082} C_VEL
LIN {X 0,Y 438.311,Z 402.457,A -85,B 0,C 180,E1 -9090.001,E2 -9090.001} C_VEL
LIN {X 0,Y 438.306,Z 402.144,A -85,B 0,C 180,E1 -9090.92,E2 -9090.92} C_VEL
LIN {X 0,Y 438.32,Z 401.294,A -85,B 0,C 180,E1 -9091.839,E2 -9091.839} C_VEL
LIN {X 0,Y 438.387,Z 399.968,A -85,B 0,C 180,E1 -9092.758,E2 -9092.758} C_VEL
LIN {X 0,Y 438.326,Z 396.968,A -85,B 0,C 180,E1 -9094.139,E2 -9094.139} C_VEL
LIN {X 0,Y 438.439,Z 392.689,A -85,B 0,C 180,E1 -9095.52,E2 -9095.52} C_VEL
LIN {X 0,Y 438.664,Z 386.756,A -85,B 0,C 180,E1 -9096.902,E2 -9096.902} C_VEL
LIN {X 0,Y 438.769,Z 381.821,A -85,B 0,C 180,E1 -9097.826,E2 -9097.826} C_VEL
LIN {X 0,Y 439.007,Z 375.874,A -85,B 0,C 180,E1 -9098.749,E2 -9098.749} C_VEL
LIN {X 0,Y 439.334,Z 368.634,A -85,B 0,C 180,E1 -9099.671,E2 -9099.671} C_VEL
LIN {X 0,Y 439.655,Z 360.901,A -85,B 0,C 180,E1 -9100.478,E2 -9100.478} C_VEL
LIN {X 0,Y 440.086,Z 352.786,A -85,B 0,C 180,E1 -9101.166,E2 -9101.166} C_VEL
LIN {X 0,Y 440.355,Z 344.352,A -85,B 0,C 180,E1 -9101.742,E2 -9101.742} C_VEL
LIN {X 0,Y 440.201,Z 338.916,A -85,B 0,C 180,E1 -9102.058,E2 -9102.058} C_VEL
LIN {X 0,Y 439.353,Z 328.872,A -85,B 0,C 180,E1 -9102.518,E2 -9102.518} C_VEL
LIN {X 0,Y 438.498,Z 320.787,A -85,B 0,C 180,E1 -9102.794,E2 -9102.794} C_VEL
LIN {X 0,Y 438.676,Z 312.354,A -85,B 0,C 180,E1 -9106,E2 -9106} C_VEL
LIN {X 0,Y 438.861,Z 304.26,A -85,B 0,C 180,E1 -9109.118,E2 -9109.118} C_VEL
LIN {X 0,Y 439.239,Z 295.401,A -85,B 0,C 180,E1 -9112.583,E2 -9112.583} C_VEL
LIN {X 0,Y 439.634,Z 286.808,A -85,B 0,C 180,E1 -9116.024,E2 -9116.024} C_VEL
LIN {X 0,Y 440.065,Z 279.201,A -85,B 0,C 180,E1 -9119.151,E2 -9119.151} C_VEL
LIN {X 0,Y 440.511,Z 271.834,A -85,B 0,C 180,E1 -9122.266,E2 -9122.266} C_VEL
LIN {X 0,Y 440.326,Z 268.003,A -85,B 0,C 180,E1 -9123.962,E2 -9123.962} C_VEL
LIN {X 0,Y 439.388,Z 262.569,A -85,B 0,C 180,E1 -9126.585,E2 -9126.585} C_VEL
LIN {X 0,Y 439.41,Z 262.565,A -85,B 0,C 180,E1 -9129.849,E2 -9129.849} C_VEL
LIN {X 0,Y 439.389,Z 262.566,A -85,B 0,C 180,E1 -9132.627,E2 -9132.627} C_VEL
LIN {X 0,Y 439.407,Z 262.563,A -85,B 0,C 180,E1 -9135.27,E2 -9135.27} C_VEL
LIN {X 0,Y 439.397,Z 262.564,A -85,B 0,C 180,E1 -9138.743,E2 -9138.743} C_VEL
LIN {X 0,Y 439.377,Z 262.57,A -85,B 0,C 180,E1 -9141.609,E2 -9141.609} C_VEL
LIN {X 0,Y 439.407,Z 262.563,A -85,B 0,C 180,E1 -9144.844,E2 -9144.844} C_VEL
LIN {X 0,Y 439.381,Z 262.568,A -85,B 0,C 180,E1 -9148.139,E2 -9148.139} C_VEL
LIN {X 0,Y 439.442,Z 262.562,A -85,B 0,C 180,E1 -9151.598,E2 -9151.598} C_VEL
LIN {X 0,Y 439.406,Z 262.563,A -85,B 0,C 180,E1 -9154.414,E2 -9154.414} C_VEL
LIN {X 0,Y 439.373,Z 262.57,A -85,B 0,C 180,E1 -9157.424,E2 -9157.424} C_VEL
LIN {X 0,Y 439.45,Z 262.558,A -85,B 0,C 180,E1 -9160.662,E2 -9160.662} C_VEL
LIN {X 0,Y 439.471,Z 262.555,A -85,B 0,C 180,E1 -9164.223,E2 -9164.223} C_VEL
LIN {X 0,Y 439.491,Z 262.553,A -85,B 0,C 180,E1 -9168,E2 -9168} C_VEL
LIN {X 0,Y 439.511,Z 262.55,A -85,B 0,C 180,E1 -9171.724,E2 -9171.724} C_VEL
LIN {X 0,Y 439.622,Z 262.538,A -85,B 0,C 180,E1 -9174.494,E2 -9174.494} C_VEL
LIN {X 0,Y 439.64,Z 262.536,A -85,B 0,C 180,E1 -9178.166,E2 -9178.166} C_VEL
LIN {X 0,Y 439.768,Z 262.519,A -85,B 0,C 180,E1 -9179.998,E2 -9179.998} C_VEL
LIN {X 0,Y 439.66,Z 262.535,A -85,B 0,C 180,E1 -9182.747,E2 -9182.747} C_VEL
LIN {X 0,Y 439.623,Z 262.539,A -85,B 0,C 180,E1 -9186.423,E2 -9186.423} C_VEL
LIN {X 0,Y 439.504,Z 262.551,A -85,B 0,C 180,E1 -9189.2,E2 -9189.2} C_VEL
LIN {X 0,Y 439.468,Z 262.556,A -85,B 0,C 180,E1 -9192.936,E2 -9192.936} C_VEL
LIN {X 0,Y 439.449,Z 262.56,A -85,B 0,C 180,E1 -9196.347,E2 -9196.347} C_VEL
LIN {X 0,Y 439.403,Z 262.566,A -85,B 0,C 180,E1 -9199.624,E2 -9199.624} C_VEL
LIN {X 0,Y 439.365,Z 262.569,A -85,B 0,C 180,E1 -9202.573,E2 -9202.573} C_VEL
LIN {X 0,Y 439.404,Z 262.566,A -85,B 0,C 180,E1 -9205.583,E2 -9205.583} C_VEL
LIN {X 0,Y 439.415,Z 262.561,A -85,B 0,C 180,E1 -9208.671,E2 -9208.671} C_VEL
LIN {X 0,Y 439.367,Z 262.571,A -85,B 0,C 180,E1 -9212.028,E2 -9212.028} C_VEL
LIN {X 0,Y 439.391,Z 262.568,A -85,B 0,C 180,E1 -9215.338,E2 -9215.338} C_VEL
LIN {X 0,Y 439.391,Z 262.565,A -85,B 0,C 180,E1 -9218.591,E2 -9218.591} C_VEL
LIN {X 0,Y 439.398,Z 262.567,A -85,B 0,C 180,E1 -9221.257,E2 -9221.257} C_VEL
LIN {X 0,Y 439.402,Z 262.565,A -85,B 0,C 180,E1 -9224.726,E2 -9224.726} C_VEL
LIN {X 0,Y 439.403,Z 262.564,A -85,B 0,C 180,E1 -9227.795,E2 -9227.795} C_VEL
LIN {X 0,Y 439.442,Z 262.558,A -85,B 0,C 180,E1 -9230.228,E2 -9230.228} C_VEL
LIN {X 0,Y 439.366,Z 262.568,A -85,B 0,C 180,E1 -9233.711,E2 -9233.711} C_VEL
LIN {X 0,Y 439.36,Z 262.571,A -85,B 0,C 180,E1 -9237.052,E2 -9237.052} C_VEL
LIN {X 0,Y 439.383,Z 262.567,A -85,B 0,C 180,E1 -9240.273,E2 -9240.273} C_VEL
LIN {X 0,Y 439.419,Z 262.562,A -85,B 0,C 180,E1 -9243.587,E2 -9243.587} C_VEL
LIN {X 0,Y 439.379,Z 262.569,A -85,B 0,C 180,E1 -9246.428,E2 -9246.428} C_VEL
LIN {X 0,Y 439.391,Z 262.565,A -85,B 0,C 180,E1 -9249.396,E2 -9249.396} C_VEL
LIN {X 0,Y 439.347,Z 262.57,A -85,B 0,C 180,E1 -9251.34,E2 -9251.34} C_VEL
LIN {X 0,Y 439.032,Z 262.613,A -85,B 0,C 180,E1 -9254.208,E2 -9254.208} C_VEL
LIN {X 0,Y 438.874,Z 262.927,A -85,B 0,C 180,E1 -9255.153,E2 -9255.153} C_VEL
LIN {X 0,Y 438.924,Z 266.389,A -85,B 0,C 180,E1 -9257.985,E2 -9257.985} C_VEL
LIN {X 0,Y 438.794,Z 271.044,A -85,B 0,C 180,E1 -9261.711,E2 -9261.711} C_VEL
LIN {X 0,Y 438.849,Z 273.398,A -85,B 0,C 180,E1 -9263.562,E2 -9263.562} C_VEL
LIN {X 0,Y 438.743,Z 276.929,A -85,B 0,C 180,E1 -9266.325,E2 -9266.325} C_VEL
LIN {X 0,Y 438.422,Z 281.722,A -85,B 0,C 180,E1 -9269.999,E2 -9269.999} C_VEL
LIN {X 0,Y 438.416,Z 282.644,A -85,B 0,C 180,E1 -9270.703,E2 -9270.703} C_VEL
LIN {X 0,Y 438.344,Z 283.852,A -85,B 0,C 180,E1 -9271.034,E2 -9271.034} C_VEL
LIN {X 0,Y 438.035,Z 286.992,A -85,B 0,C 180,E1 -9271.374,E2 -9271.374} C_VEL
LIN {X 0,Y 437.653,Z 290.268,A -85,B 0,C 180,E1 -9271.548,E2 -9271.548} C_VEL
LIN {X 0,Y 436.182,Z 298.528,A -85,B 0,C 180,E1 -9271.888,E2 -9271.888} C_VEL
LIN {X 0,Y 434.201,Z 306.225,A -85,B 0,C 180,E1 -9272.272,E2 -9272.272} C_VEL
LIN {X 0,Y 433.511,Z 310.65,A -85,B 0,C 180,E1 -9272.583,E2 -9272.583} C_VEL
LIN {X 0,Y 433.178,Z 318.789,A -85,B 0,C 180,E1 -9273.254,E2 -9273.254} C_VEL
LIN {X 0,Y 432.765,Z 326.83,A -85,B 0,C 180,E1 -9274.073,E2 -9274.073} C_VEL
LIN {X 0,Y 432.521,Z 333.438,A -85,B 0,C 180,E1 -9274.892,E2 -9274.892} C_VEL
LIN {X 0,Y 432.156,Z 339.743,A -85,B 0,C 180,E1 -9275.832,E2 -9275.832} C_VEL
LIN {X 0,Y 432.008,Z 345.201,A -85,B 0,C 180,E1 -9276.822,E2 -9276.822} C_VEL
LIN {X 0,Y 431.728,Z 350.285,A -85,B 0,C 180,E1 -9277.952,E2 -9277.952} C_VEL
LIN {X 0,Y 431.521,Z 353.72,A -85,B 0,C 180,E1 -9278.899,E2 -9278.899} C_VEL
LIN {X 0,Y 431.413,Z 356.509,A -85,B 0,C 180,E1 -9279.848,E2 -9279.848} C_VEL
LIN {X 0,Y 431.292,Z 359.548,A -85,B 0,C 180,E1 -9281.275,E2 -9281.275} C_VEL
LIN {X 0,Y 431.251,Z 360.901,A -85,B 0,C 180,E1 -9282.23,E2 -9282.23} C_VEL
LIN {X 0,Y 431.191,Z 361.759,A -85,B 0,C 180,E1 -9283.189,E2 -9283.189} C_VEL
LIN {X 0,Y 431.183,Z 362.084,A -85,B 0,C 180,E1 -9284.15,E2 -9284.15} C_VEL
LIN {X 0,Y 431.22,Z 361.807,A -85,B 0,C 180,E1 -9285.114,E2 -9285.114} C_VEL
LIN {X 0,Y 431.292,Z 361.019,A -85,B 0,C 180,E1 -9286.081,E2 -9286.081} C_VEL
LIN {X 0,Y 431.369,Z 359.714,A -85,B 0,C 180,E1 -9287.052,E2 -9287.052} C_VEL
LIN {X 0,Y 431.544,Z 356.671,A -85,B 0,C 180,E1 -9288.515,E2 -9288.515} C_VEL
LIN {X 0,Y 431.828,Z 352.246,A -85,B 0,C 180,E1 -9289.984,E2 -9289.984} C_VEL
LIN {X 0,Y 432.078,Z 347.189,A -85,B 0,C 180,E1 -9291.216,E2 -9291.216} C_VEL
LIN {X 0,Y 432.468,Z 340.879,A -85,B 0,C 180,E1 -9292.418,E2 -9292.418} C_VEL
LIN {X 0,Y 432.865,Z 334.251,A -85,B 0,C 180,E1 -9293.438,E2 -9293.438} C_VEL
LIN {X 0,Y 433.147,Z 328.655,A -85,B 0,C 180,E1 -9294.161,E2 -9294.161} C_VEL
LIN {X 0,Y 433.524,Z 321.591,A -85,B 0,C 180,E1 -9294.927,E2 -9294.927} C_VEL
LIN {X 0,Y 434.001,Z 313.184,A -85,B 0,C 180,E1 -9295.668,E2 -9295.668} C_VEL
LIN {X 0,Y 434.317,Z 305.817,A -85,B 0,C 180,E1 -9296.195,E2 -9296.195} C_VEL
LIN {X 0,Y 434.324,Z 298.649,A -85,B 0,C 180,E1 -9296.624,E2 -9296.624} C_VEL
LIN {X 0,Y 432.581,Z 289.466,A -85,B 0,C 180,E1 -9297.108,E2 -9297.108} C_VEL
LIN {X 0,Y 431.382,Z 284.045,A -85,B 0,C 180,E1 -9297.352,E2 -9297.352} C_VEL
LIN {X 0,Y 431.498,Z 280.315,A -85,B 0,C 180,E1 -9300.324,E2 -9300.324} C_VEL
LIN {X 0,Y 431.548,Z 276.007,A -85,B 0,C 180,E1 -9303.848,E2 -9303.848} C_VEL
LIN {X 0,Y 431.683,Z 272.113,A -85,B 0,C 180,E1 -9307.089,E2 -9307.089} C_VEL
LIN {X 0,Y 431.787,Z 267.996,A -85,B 0,C 180,E1 -9310.62,E2 -9310.62} C_VEL
LIN {X 0,Y 431.926,Z 265.123,A -85,B 0,C 180,E1 -9313.107,E2 -9313.107} C_VEL
LIN {X 0,Y 431.971,Z 263.679,A -85,B 0,C 180,E1 -9314.392,E2 -9314.392} C_VEL
LIN {X 0,Y 432.224,Z 263.456,A -85,B 0,C 180,E1 -9317.027,E2 -9317.027} C_VEL
LIN {X 0,Y 432.334,Z 263.446,A -85,B 0,C 180,E1 -9319.818,E2 -9319.818} C_VEL
LIN {X 0,Y 432.298,Z 263.451,A -85,B 0,C 180,E1 -9323.024,E2 -9323.024} C_VEL
LIN {X 0,Y 432.34,Z 263.446,A -85,B 0,C 180,E1 -9325.997,E2 -9325.997} C_VEL
LIN {X 0,Y 432.328,Z 263.445,A -85,B 0,C 180,E1 -9329.491,E2 -9329.491} C_VEL
LIN {X 0,Y 432.374,Z 263.438,A -85,B 0,C 180,E1 -9332.93,E2 -9332.93} C_VEL
LIN {X 0,Y 432.352,Z 263.439,A -85,B 0,C 180,E1 -9336.025,E2 -9336.025} C_VEL
LIN {X 0,Y 432.333,Z 263.442,A -85,B 0,C 180,E1 -9339.047,E2 -9339.047} C_VEL
LIN {X 0,Y 432.362,Z 263.439,A -85,B 0,C 180,E1 -9342.013,E2 -9342.013} C_VEL
LIN {X 0,Y 432.38,Z 263.439,A -85,B 0,C 180,E1 -9344.928,E2 -9344.928} C_VEL
LIN {X 0,Y 432.467,Z 263.429,A -85,B 0,C 180,E1 -9347.806,E2 -9347.806} C_VEL
LIN {X 0,Y 432.469,Z 263.428,A -85,B 0,C 180,E1 -9351.592,E2 -9351.592} C_VEL
LIN {X 0,Y 432.572,Z 263.415,A -85,B 0,C 180,E1 -9354.408,E2 -9354.408} C_VEL
LIN {X 0,Y 432.596,Z 263.408,A -85,B 0,C 180,E1 -9358.14,E2 -9358.14} C_VEL
LIN {X 0,Y 432.721,Z 263.395,A -85,B 0,C 180,E1 -9360.002,E2 -9360.002} C_VEL
LIN {X 0,Y 432.581,Z 263.412,A -85,B 0,C 180,E1 -9362.795,E2 -9362.795} C_VEL
LIN {X 0,Y 432.563,Z 263.412,A -85,B 0,C 180,E1 -9366.532,E2 -9366.532} C_VEL
LIN {X 0,Y 432.432,Z 263.431,A -85,B 0,C 180,E1 -9369.355,E2 -9369.355} C_VEL
LIN {X 0,Y 432.436,Z 263.431,A -85,B 0,C 180,E1 -9372.813,E2 -9372.813} C_VEL
LIN {X 0,Y 432.403,Z 263.439,A -85,B 0,C 180,E1 -9376.48,E2 -9376.48} C_VEL
LIN {X 0,Y 432.33,Z 263.446,A -85,B 0,C 180,E1 -9379.962,E2 -9379.962} C_VEL
LIN {X 0,Y 432.311,Z 263.451,A -85,B 0,C 180,E1 -9382.966,E2 -9382.966} C_VEL
LIN {X 0,Y 432.333,Z 263.445,A -85,B 0,C 180,E1 -9385.004,E2 -9385.004} C_VEL
LIN {X 0,Y 432.34,Z 263.445,A -85,B 0,C 180,E1 -9388.127,E2 -9388.127} C_VEL
LIN {X 0,Y 432.315,Z 263.449,A -85,B 0,C 180,E1 -9391.348,E2 -9391.348} C_VEL
LIN {X 0,Y 432.333,Z 263.447,A -85,B 0,C 180,E1 -9394.679,E2 -9394.679} C_VEL
LIN {X 0,Y 432.338,Z 263.445,A -85,B 0,C 180,E1 -9398.151,E2 -9398.151} C_VEL
LIN {X 0,Y 432.362,Z 263.443,A -85,B 0,C 180,E1 -9401.609,E2 -9401.609} C_VEL
LIN {X 0,Y 432.33,Z 263.448,A -85,B 0,C 180,E1 -9404.349,E2 -9404.349} C_VEL
LIN {X 0,Y 432.316,Z 263.451,A -85,B 0,C 180,E1 -9407.017,E2 -9407.017} C_VEL
LIN {X 0,Y 432.33,Z 263.448,A -85,B 0,C 180,E1 -9409.822,E2 -9409.822} C_VEL
LIN {X 0,Y 432.354,Z 263.537,A -85,B 0,C 180,E1 -9411.783,E2 -9411.783} C_VEL
LIN {X 0,Y 433.606,Z 270.443,A -85,B 0,C 180,E1 -9415.44,E2 -9415.44} C_VEL
LIN {X 0,Y 433.885,Z 274.366,A -85,B 0,C 180,E1 -9417.384,E2 -9417.384} C_VEL
LIN {X 0,Y 433.356,Z 280.854,A -85,B 0,C 180,E1 -9420.356,E2 -9420.356} C_VEL
LIN {X 0,Y 432.832,Z 287.467,A -85,B 0,C 180,E1 -9423.26,E2 -9423.26} C_VEL
LIN {X 0,Y 432.368,Z 295.146,A -85,B 0,C 180,E1 -9426.533,E2 -9426.533} C_VEL
LIN {X 0,Y 431.936,Z 303.593,A -85,B 0,C 180,E1 -9430.022,E2 -9430.022} C_VEL
LIN {X 0,Y 431.668,Z 312.231,A -85,B 0,C 180,E1 -9433.496,E2 -9433.496} C_VEL
LIN {X 0,Y 431.444,Z 320.406,A -85,B 0,C 180,E1 -9436.654,E2 -9436.654} C_VEL
LIN {X 0,Y 433.127,Z 332.571,A -85,B 0,C 180,E1 -9437.141,E2 -9437.141} C_VEL
LIN {X 0,Y 433.796,Z 343.2,A -85,B 0,C 180,E1 -9437.736,E2 -9437.736} C_VEL
LIN {X 0,Y 433.476,Z 351.539,A -85,B 0,C 180,E1 -9438.309,E2 -9438.309} C_VEL
LIN {X 0,Y 433.03,Z 359.73,A -85,B 0,C 180,E1 -9439.008,E2 -9439.008} C_VEL
LIN {X 0,Y 432.568,Z 367.522,A -85,B 0,C 180,E1 -9439.824,E2 -9439.824} C_VEL
LIN {X 0,Y 432.241,Z 373.975,A -85,B 0,C 180,E1 -9440.644,E2 -9440.644} C_VEL
LIN {X 0,Y 431.863,Z 380.134,A -85,B 0,C 180,E1 -9441.579,E2 -9441.579} C_VEL
LIN {X 0,Y 431.563,Z 386.435,A -85,B 0,C 180,E1 -9442.751,E2 -9442.751} C_VEL
LIN {X 0,Y 431.363,Z 391.462,A -85,B 0,C 180,E1 -9443.924,E2 -9443.924} C_VEL
LIN {X 0,Y 431.299,Z 396.006,A -85,B 0,C 180,E1 -9445.328,E2 -9445.328} C_VEL
LIN {X 0,Y 431.236,Z 398.319,A -85,B 0,C 180,E1 -9446.264,E2 -9446.264} C_VEL
LIN {X 0,Y 431.295,Z 400.004,A -85,B 0,C 180,E1 -9447.199,E2 -9447.199} C_VEL
LIN {X 0,Y 431.242,Z 401.177,A -85,B 0,C 180,E1 -9448.133,E2 -9448.133} C_VEL
LIN {X 0,Y 431.219,Z 401.878,A -85,B 0,C 180,E1 -9449.067,E2 -9449.067} C_VEL
LIN {X 0,Y 431.222,Z 402.118,A -85,B 0,C 180,E1 -9450.001,E2 -9450.001} C_VEL
LIN {X 0,Y 431.219,Z 401.803,A -85,B 0,C 180,E1 -9450.935,E2 -9450.935} C_VEL
LIN {X 0,Y 431.243,Z 400.933,A -85,B 0,C 180,E1 -9451.869,E2 -9451.869} C_VEL
LIN {X 0,Y 431.315,Z 399.586,A -85,B 0,C 180,E1 -9452.803,E2 -9452.803} C_VEL
LIN {X 0,Y 431.243,Z 396.563,A -85,B 0,C 180,E1 -9454.207,E2 -9454.207} C_VEL
LIN {X 0,Y 431.341,Z 392.253,A -85,B 0,C 180,E1 -9455.611,E2 -9455.611} C_VEL
LIN {X 0,Y 431.594,Z 386.27,A -85,B 0,C 180,E1 -9457.016,E2 -9457.016} C_VEL
LIN {X 0,Y 431.705,Z 381.302,A -85,B 0,C 180,E1 -9457.955,E2 -9457.955} C_VEL
LIN {X 0,Y 431.972,Z 375.318,A -85,B 0,C 180,E1 -9458.892,E2 -9458.892} C_VEL
LIN {X 0,Y 432.295,Z 368.031,A -85,B 0,C 180,E1 -9459.83,E2 -9459.83} C_VEL
LIN {X 0,Y 432.648,Z 360.244,A -85,B 0,C 180,E1 -9460.649,E2 -9460.649} C_VEL
LIN {X 0,Y 433.09,Z 352.056,A -85,B 0,C 180,E1 -9461.349,E2 -9461.349} C_VEL
LIN {X 0,Y 433.371,Z 343.524,A -85,B 0,C 180,E1 -9461.934,E2 -9461.934} C_VEL
LIN {X 0,Y 432.803,Z 334.301,A -85,B 0,C 180,E1 -9462.442,E2 -9462.442} C_VEL
LIN {X 0,Y 431.574,Z 322.179,A -85,B 0,C 180,E1 -9462.929,E2 -9462.929} C_VEL
LIN {X 0,Y 431.4,Z 320.473,A -85,B 0,C 180,E1 -9462.974,E2 -9462.974} C_VEL
LIN {X 0,Y 431.604,Z 312.4,A -85,B 0,C 180,E1 -9466.11,E2 -9466.11} C_VEL
LIN {X 0,Y 431.809,Z 304.363,A -85,B 0,C 180,E1 -9469.265,E2 -9469.265} C_VEL
LIN {X 0,Y 432.158,Z 296.337,A -85,B 0,C 180,E1 -9472.469,E2 -9472.469} C_VEL
LIN {X 0,Y 432.567,Z 287.603,A -85,B 0,C 180,E1 -9476.02,E2 -9476.02} C_VEL
LIN {X 0,Y 433.115,Z 278.912,A -85,B 0,C 180,E1 -9479.665,E2 -9479.665} C_VEL
LIN {X 0,Y 433.508,Z 272.26,A -85,B 0,C 180,E1 -9482.538,E2 -9482.538} C_VEL
LIN {X 0,Y 433.262,Z 268.653,A -85,B 0,C 180,E1 -9484.179,E2 -9484.179} C_VEL
LIN {X 0,Y 432.358,Z 263.444,A -85,B 0,C 180,E1 -9486.683,E2 -9486.683} C_VEL
LIN {X 0,Y 432.342,Z 263.446,A -85,B 0,C 180,E1 -9490.179,E2 -9490.179} C_VEL
LIN {X 0,Y 432.325,Z 263.444,A -85,B 0,C 180,E1 -9493.061,E2 -9493.061} C_VEL
LIN {X 0,Y 432.342,Z 263.446,A -85,B 0,C 180,E1 -9495.665,E2 -9495.665} C_VEL
LIN {X 0,Y 432.341,Z 263.444,A -85,B 0,C 180,E1 -9498.398,E2 -9498.398} C_VEL
LIN {X 0,Y 432.341,Z 263.446,A -85,B 0,C 180,E1 -9501.849,E2 -9501.849} C_VEL
LIN {X 0,Y 432.348,Z 263.444,A -85,B 0,C 180,E1 -9505.322,E2 -9505.322} C_VEL
LIN {X 0,Y 432.33,Z 263.445,A -85,B 0,C 180,E1 -9508.653,E2 -9508.653} C_VEL
LIN {X 0,Y 432.391,Z 263.438,A -85,B 0,C 180,E1 -9511.876,E2 -9511.876} C_VEL
LIN {X 0,Y 432.355,Z 263.444,A -85,B 0,C 180,E1 -9514.998,E2 -9514.998} C_VEL
LIN {X 0,Y 432.366,Z 263.44,A -85,B 0,C 180,E1 -9518.045,E2 -9518.045} C_VEL
LIN {X 0,Y 432.393,Z 263.439,A -85,B 0,C 180,E1 -9521.029,E2 -9521.029} C_VEL
LIN {X 0,Y 432.439,Z 263.431,A -85,B 0,C 180,E1 -9523.96,E2 -9523.96} C_VEL
LIN {X 0,Y 432.467,Z 263.428,A -85,B 0,C 180,E1 -9527.802,E2 -9527.802} C_VEL
LIN {X 0,Y 432.471,Z 263.428,A -85,B 0,C 180,E1 -9531.588,E2 -9531.588} C_VEL
LIN {X 0,Y 432.598,Z 263.413,A -85,B 0,C 180,E1 -9534.405,E2 -9534.405} C_VEL
LIN {X 0,Y 432.609,Z 263.411,A -85,B 0,C 180,E1 -9538.136,E2 -9538.136} C_VEL
LIN {X 0,Y 432.738,Z 263.394,A -85,B 0,C 180,E1 -9539.998,E2 -9539.998} C_VEL
LIN {X 0,Y 432.61,Z 263.413,A -85,B 0,C 180,E1 -9542.792,E2 -9542.792} C_VEL
LIN {X 0,Y 432.577,Z 263.416,A -85,B 0,C 180,E1 -9546.528,E2 -9546.528} C_VEL
LIN {X 0,Y 432.446,Z 263.43,A -85,B 0,C 180,E1 -9549.351,E2 -9549.351} C_VEL
LIN {X 0,Y 432.434,Z 263.433,A -85,B 0,C 180,E1 -9552.801,E2 -9552.801} C_VEL
LIN {X 0,Y 432.414,Z 263.436,A -85,B 0,C 180,E1 -9556.477,E2 -9556.477} C_VEL
LIN {X 0,Y 432.339,Z 263.446,A -85,B 0,C 180,E1 -9559.958,E2 -9559.958} C_VEL
LIN {X 0,Y 432.319,Z 263.446,A -85,B 0,C 180,E1 -9562.962,E2 -9562.962} C_VEL
LIN {X 0,Y 432.363,Z 263.444,A -85,B 0,C 180,E1 -9566.03,E2 -9566.03} C_VEL
LIN {X 0,Y 432.34,Z 263.444,A -85,B 0,C 180,E1 -9569.185,E2 -9569.185} C_VEL
LIN {X 0,Y 432.319,Z 263.446,A -85,B 0,C 180,E1 -9572.441,E2 -9572.441} C_VEL
LIN {X 0,Y 432.341,Z 263.446,A -85,B 0,C 180,E1 -9575.63,E2 -9575.63} C_VEL
LIN {X 0,Y 432.36,Z 263.444,A -85,B 0,C 180,E1 -9579.339,E2 -9579.339} C_VEL
LIN {X 0,Y 432.367,Z 263.442,A -85,B 0,C 180,E1 -9581.79,E2 -9581.79} C_VEL
LIN {X 0,Y 432.37,Z 263.439,A -85,B 0,C 180,E1 -9584.339,E2 -9584.339} C_VEL
LIN {X 0,Y 432.357,Z 263.444,A -85,B 0,C 180,E1 -9587.007,E2 -9587.007} C_VEL
LIN {X 0,Y 432.348,Z 263.442,A -85,B 0,C 180,E1 -9589.814,E2 -9589.814} C_VEL
LIN {X 0,Y 432.307,Z 263.45,A -85,B 0,C 180,E1 -9593.021,E2 -9593.021} C_VEL
LIN {X 0,Y 432.347,Z 263.442,A -85,B 0,C 180,E1 -9595.994,E2 -9595.994} C_VEL
LIN {X 0,Y 432.382,Z 263.438,A -85,B 0,C 180,E1 -9599.742,E2 -9599.742} C_VEL
LIN {X 0,Y 432.386,Z 263.439,A -85,B 0,C 180,E1 -9603.37,E2 -9603.37} C_VEL
LIN {X 0,Y 432.36,Z 263.442,A -85,B 0,C 180,E1 -9606.022,E2 -9606.022} C_VEL
LIN {X 0,Y 432.358,Z 263.442,A -85,B 0,C 180,E1 -9609.045,E2 -9609.045} C_VEL
LIN {X 0,Y 432.333,Z 263.445,A -85,B 0,C 180,E1 -9611.026,E2 -9611.026} C_VEL
LIN {X 0,Y 432.017,Z 263.486,A -85,B 0,C 180,E1 -9613.944,E2 -9613.944} C_VEL
LIN {X 0,Y 431.849,Z 263.508,A -85,B 0,C 180,E1 -9614.906,E2 -9614.906} C_VEL
LIN {X 0,Y 431.889,Z 266.844,A -85,B 0,C 180,E1 -9617.786,E2 -9617.786} C_VEL
LIN {X 0,Y 431.746,Z 271.54,A -85,B 0,C 180,E1 -9621.575,E2 -9621.575} C_VEL
LIN {X 0,Y 431.778,Z 273.885,A -85,B 0,C 180,E1 -9623.456,E2 -9623.456} C_VEL
LIN {X 0,Y 431.677,Z 277.453,A -85,B 0,C 180,E1 -9626.265,E2 -9626.265} C_VEL
LIN {X 0,Y 431.356,Z 282.276,A -85,B 0,C 180,E1 -9629.999,E2 -9629.999} C_VEL
LIN {X 0,Y 431.344,Z 283.762,A -85,B 0,C 180,E1 -9631.137,E2 -9631.137} C_VEL
LIN {X 0,Y 433.46,Z 295.777,A -85,B 0,C 180,E1 -9631.683,E2 -9631.683} C_VEL
LIN {X 0,Y 433.838,Z 300.259,A -85,B 0,C 180,E1 -9631.913,E2 -9631.913} C_VEL
LIN {X 0,Y 433.511,Z 310.65,A -85,B 0,C 180,E1 -9632.583,E2 -9632.583} C_VEL
LIN {X 0,Y 432.643,Z 315.878,A -85,B 0,C 180,E1 -9632.974,E2 -9632.974} C_VEL
LIN {X 0,Y 429.428,Z 323.859,A -85,B 0,C 180,E1 -9633.655,E2 -9633.655} C_VEL
LIN {X 0,Y 426.278,Z 331.083,A -85,B 0,C 180,E1 -9634.423,E2 -9634.423} C_VEL
LIN {X 0,Y 425.434,Z 335.158,A -85,B 0,C 180,E1 -9634.972,E2 -9634.972} C_VEL
LIN {X 0,Y 425.046,Z 342.655,A -85,B 0,C 180,E1 -9636.169,E2 -9636.169} C_VEL
LIN {X 0,Y 424.866,Z 347.863,A -85,B 0,C 180,E1 -9637.215,E2 -9637.215} C_VEL
LIN {X 0,Y 424.515,Z 353.151,A -85,B 0,C 180,E1 -9638.568,E2 -9638.568} C_VEL
LIN {X 0,Y 424.378,Z 356.152,A -85,B 0,C 180,E1 -9639.531,E2 -9639.531} C_VEL
LIN {X 0,Y 424.293,Z 358.49,A -85,B 0,C 180,E1 -9640.497,E2 -9640.497} C_VEL
LIN {X 0,Y 424.181,Z 361.176,A -85,B 0,C 180,E1 -9642.182,E2 -9642.182} C_VEL
LIN {X 0,Y 424.103,Z 362.159,A -85,B 0,C 180,E1 -9643.413,E2 -9643.413} C_VEL
LIN {X 0,Y 424.092,Z 362.39,A -85,B 0,C 180,E1 -9644.392,E2 -9644.392} C_VEL
LIN {X 0,Y 424.14,Z 362.066,A -85,B 0,C 180,E1 -9645.373,E2 -9645.373} C_VEL
LIN {X 0,Y 424.219,Z 361.146,A -85,B 0,C 180,E1 -9646.357,E2 -9646.357} C_VEL
LIN {X 0,Y 424.365,Z 358.851,A -85,B 0,C 180,E1 -9647.84,E2 -9647.84} C_VEL
LIN {X 0,Y 424.64,Z 354.922,A -85,B 0,C 180,E1 -9649.382,E2 -9649.382} C_VEL
LIN {X 0,Y 424.927,Z 349.813,A -85,B 0,C 180,E1 -9650.828,E2 -9650.828} C_VEL
LIN {X 0,Y 425.341,Z 343.523,A -85,B 0,C 180,E1 -9652.191,E2 -9652.191} C_VEL
LIN {X 0,Y 425.763,Z 336.677,A -85,B 0,C 180,E1 -9653.337,E2 -9653.337} C_VEL
LIN {X 0,Y 426.198,Z 329.172,A -85,B 0,C 180,E1 -9654.345,E2 -9654.345} C_VEL
LIN {X 0,Y 426.625,Z 322.116,A -85,B 0,C 180,E1 -9655.125,E2 -9655.125} C_VEL
LIN {X 0,Y 427.095,Z 314.074,A -85,B 0,C 180,E1 -9655.852,E2 -9655.852} C_VEL
LIN {X 0,Y 427.454,Z 306.175,A -85,B 0,C 180,E1 -9656.43,E2 -9656.43} C_VEL
LIN {X 0,Y 427.635,Z 301.214,A -85,B 0,C 180,E1 -9656.744,E2 -9656.744} C_VEL
LIN {X 0,Y 425.786,Z 290.842,A -85,B 0,C 180,E1 -9657.32,E2 -9657.32} C_VEL
LIN {X 0,Y 424.334,Z 284.37,A -85,B 0,C 180,E1 -9657.628,E2 -9657.628} C_VEL
LIN {X 0,Y 424.437,Z 280.343,A -85,B 0,C 180,E1 -9660.883,E2 -9660.883} C_VEL
LIN {X 0,Y 424.485,Z 276.261,A -85,B 0,C 180,E1 -9664.256,E2 -9664.256} C_VEL
LIN {X 0,Y 424.627,Z 272.568,A -85,B 0,C 180,E1 -9667.401,E2 -9667.401} C_VEL
LIN {X 0,Y 424.74,Z 269.031,A -85,B 0,C 180,E1 -9670.439,E2 -9670.439} C_VEL
LIN {X 0,Y 424.923,Z 265.01,A -85,B 0,C 180,E1 -9673.998,E2 -9673.998} C_VEL
LIN {X 0,Y 424.952,Z 264.366,A -85,B 0,C 180,E1 -9674.675,E2 -9674.675} C_VEL
LIN {X 0,Y 425.179,Z 264.333,A -85,B 0,C 180,E1 -9677.338,E2 -9677.338} C_VEL
LIN {X 0,Y 425.287,Z 264.323,A -85,B 0,C 180,E1 -9679.876,E2 -9679.876} C_VEL
LIN {X 0,Y 425.267,Z 264.328,A -85,B 0,C 180,E1 -9682.488,E2 -9682.488} C_VEL
LIN {X 0,Y 425.288,Z 264.325,A -85,B 0,C 180,E1 -9685.818,E2 -9685.818} C_VEL
LIN {X 0,Y 425.271,Z 264.326,A -85,B 0,C 180,E1 -9689.24,E2 -9689.24} C_VEL
LIN {X 0,Y 425.331,Z 264.318,A -85,B 0,C 180,E1 -9692.444,E2 -9692.444} C_VEL
LIN {X 0,Y 425.332,Z 264.316,A -85,B 0,C 180,E1 -9695.603,E2 -9695.603} C_VEL
LIN {X 0,Y 425.276,Z 264.323,A -85,B 0,C 180,E1 -9698.683,E2 -9698.683} C_VEL
LIN {X 0,Y 425.317,Z 264.319,A -85,B 0,C 180,E1 -9701.704,E2 -9701.704} C_VEL
LIN {X 0,Y 425.333,Z 264.318,A -85,B 0,C 180,E1 -9704.672,E2 -9704.672} C_VEL
LIN {X 0,Y 425.416,Z 264.306,A -85,B 0,C 180,E1 -9707.6,E2 -9707.6} C_VEL
LIN {X 0,Y 425.423,Z 264.306,A -85,B 0,C 180,E1 -9711.451,E2 -9711.451} C_VEL
LIN {X 0,Y 425.527,Z 264.291,A -85,B 0,C 180,E1 -9714.315,E2 -9714.315} C_VEL
LIN {X 0,Y 425.565,Z 264.284,A -85,B 0,C 180,E1 -9718.109,E2 -9718.109} C_VEL
LIN {X 0,Y 425.69,Z 264.271,A -85,B 0,C 180,E1 -9720.002,E2 -9720.002} C_VEL
LIN {X 0,Y 425.535,Z 264.29,A -85,B 0,C 180,E1 -9722.842,E2 -9722.842} C_VEL
LIN {X 0,Y 425.521,Z 264.289,A -85,B 0,C 180,E1 -9726.641,E2 -9726.641} C_VEL
LIN {X 0,Y 425.391,Z 264.308,A -85,B 0,C 180,E1 -9729.511,E2 -9729.511} C_VEL
LIN {X 0,Y 425.395,Z 264.309,A -85,B 0,C 180,E1 -9732.912,E2 -9732.912} C_VEL
LIN {X 0,Y 425.352,Z 264.316,A -85,B 0,C 180,E1 -9736.606,E2 -9736.606} C_VEL
LIN {X 0,Y 425.32,Z 264.321,A -85,B 0,C 180,E1 -9739.637,E2 -9739.637} C_VEL
LIN {X 0,Y 425.28,Z 264.322,A -85,B 0,C 180,E1 -9742.34,E2 -9742.34} C_VEL
LIN {X 0,Y 425.314,Z 264.322,A -85,B 0,C 180,E1 -9744.659,E2 -9744.659} C_VEL
LIN {X 0,Y 425.265,Z 264.33,A -85,B 0,C 180,E1 -9747.565,E2 -9747.565} C_VEL
LIN {X 0,Y 425.284,Z 264.329,A -85,B 0,C 180,E1 -9750.763,E2 -9750.763} C_VEL
LIN {X 0,Y 425.305,Z 264.324,A -85,B 0,C 180,E1 -9754.29,E2 -9754.29} C_VEL
LIN {X 0,Y 425.276,Z 264.325,A -85,B 0,C 180,E1 -9757.696,E2 -9757.696} C_VEL
LIN {X 0,Y 425.295,Z 264.323,A -85,B 0,C 180,E1 -9760.525,E2 -9760.525} C_VEL
LIN {X 0,Y 425.254,Z 264.331,A -85,B 0,C 180,E1 -9763.353,E2 -9763.353} C_VEL
LIN {X 0,Y 425.253,Z 264.327,A -85,B 0,C 180,E1 -9766.651,E2 -9766.651} C_VEL
LIN {X 0,Y 425.284,Z 264.325,A -85,B 0,C 180,E1 -9769.874,E2 -9769.874} C_VEL
LIN {X 0,Y 425.335,Z 264.446,A -85,B 0,C 180,E1 -9771.486,E2 -9771.486} C_VEL
LIN {X 0,Y 426.378,Z 270.483,A -85,B 0,C 180,E1 -9774.769,E2 -9774.769} C_VEL
LIN {X 0,Y 426.897,Z 273.907,A -85,B 0,C 180,E1 -9776.531,E2 -9776.531} C_VEL
LIN {X 0,Y 426.621,Z 278.916,A -85,B 0,C 180,E1 -9778.941,E2 -9778.941} C_VEL
LIN {X 0,Y 426.046,Z 285.518,A -85,B 0,C 180,E1 -9781.959,E2 -9781.959} C_VEL
LIN {X 0,Y 425.459,Z 293.842,A -85,B 0,C 180,E1 -9785.61,E2 -9785.61} C_VEL
LIN {X 0,Y 425.008,Z 301.031,A -85,B 0,C 180,E1 -9788.668,E2 -9788.668} C_VEL
LIN {X 0,Y 424.678,Z 309.508,A -85,B 0,C 180,E1 -9792.174,E2 -9792.174} C_VEL
LIN {X 0,Y 424.461,Z 316.777,A -85,B 0,C 180,E1 -9795.131,E2 -9795.131} C_VEL
LIN {X 0,Y 424.379,Z 319.894,A -85,B 0,C 180,E1 -9796.382,E2 -9796.382} C_VEL
LIN {X 0,Y 426.062,Z 331.878,A -85,B 0,C 180,E1 -9796.867,E2 -9796.867} C_VEL
LIN {X 0,Y 426.782,Z 341.93,A -85,B 0,C 180,E1 -9797.431,E2 -9797.431} C_VEL
LIN {X 0,Y 426.635,Z 350.188,A -85,B 0,C 180,E1 -9797.998,E2 -9797.998} C_VEL
LIN {X 0,Y 426.088,Z 358.56,A -85,B 0,C 180,E1 -9798.706,E2 -9798.706} C_VEL
LIN {X 0,Y 425.627,Z 366.484,A -85,B 0,C 180,E1 -9799.536,E2 -9799.536} C_VEL
LIN {X 0,Y 425.224,Z 373.899,A -85,B 0,C 180,E1 -9800.488,E2 -9800.488} C_VEL
LIN {X 0,Y 424.755,Z 381.432,A -85,B 0,C 180,E1 -9801.677,E2 -9801.677} C_VEL
LIN {X 0,Y 424.452,Z 387.391,A -85,B 0,C 180,E1 -9802.868,E2 -9802.868} C_VEL
LIN {X 0,Y 424.266,Z 392.852,A -85,B 0,C 180,E1 -9804.297,E2 -9804.297} C_VEL
LIN {X 0,Y 424.164,Z 396.913,A -85,B 0,C 180,E1 -9805.725,E2 -9805.725} C_VEL
LIN {X 0,Y 424.191,Z 399.725,A -85,B 0,C 180,E1 -9807.152,E2 -9807.152} C_VEL
LIN {X 0,Y 424.167,Z 400.878,A -85,B 0,C 180,E1 -9808.102,E2 -9808.102} C_VEL
LIN {X 0,Y 424.136,Z 401.558,A -85,B 0,C 180,E1 -9809.052,E2 -9809.052} C_VEL
LIN {X 0,Y 424.137,Z 401.778,A -85,B 0,C 180,E1 -9810.001,E2 -9810.001} C_VEL
LIN {X 0,Y 424.136,Z 401.461,A -85,B 0,C 180,E1 -9810.951,E2 -9810.951} C_VEL
LIN {X 0,Y 424.168,Z 400.573,A -85,B 0,C 180,E1 -9811.9,E2 -9811.9} C_VEL
LIN {X 0,Y 424.225,Z 399.203,A -85,B 0,C 180,E1 -9812.85,E2 -9812.85} C_VEL
LIN {X 0,Y 424.166,Z 396.157,A -85,B 0,C 180,E1 -9814.277,E2 -9814.277} C_VEL
LIN {X 0,Y 424.248,Z 391.813,A -85,B 0,C 180,E1 -9815.706,E2 -9815.706} C_VEL
LIN {X 0,Y 424.517,Z 385.784,A -85,B 0,C 180,E1 -9817.134,E2 -9817.134} C_VEL
LIN {X 0,Y 424.639,Z 380.783,A -85,B 0,C 180,E1 -9818.088,E2 -9818.088} C_VEL
LIN {X 0,Y 424.938,Z 374.758,A -85,B 0,C 180,E1 -9819.041,E2 -9819.041} C_VEL
LIN {X 0,Y 425.253,Z 367.415,A -85,B 0,C 180,E1 -9819.994,E2 -9819.994} C_VEL
LIN {X 0,Y 425.614,Z 359.562,A -85,B 0,C 180,E1 -9820.827,E2 -9820.827} C_VEL
LIN {X 0,Y 426.084,Z 351.293,A -85,B 0,C 180,E1 -9821.538,E2 -9821.538} C_VEL
LIN {X 0,Y 426.359,Z 342.641,A -85,B 0,C 180,E1 -9822.133,E2 -9822.133} C_VEL
LIN {X 0,Y 425.399,Z 330.81,A -85,B 0,C 180,E1 -9822.771,E2 -9822.771} C_VEL
LIN {X 0,Y 424.31,Z 320.129,A -85,B 0,C 180,E1 -9823.176,E2 -9823.176} C_VEL
LIN {X 0,Y 424.537,Z 312.111,A -85,B 0,C 180,E1 -9826.347,E2 -9826.347} C_VEL
LIN {X 0,Y 424.758,Z 303.57,A -85,B 0,C 180,E1 -9829.778,E2 -9829.778} C_VEL
LIN {X 0,Y 425.14,Z 295.969,A -85,B 0,C 180,E1 -9832.861,E2 -9832.861} C_VEL
LIN {X 0,Y 425.574,Z 287.303,A -85,B 0,C 180,E1 -9836.481,E2 -9836.481} C_VEL
LIN {X 0,Y 426.152,Z 278.611,A -85,B 0,C 180,E1 -9840.2,E2 -9840.2} C_VEL
LIN {X 0,Y 426.53,Z 272.422,A -85,B 0,C 180,E1 -9842.94,E2 -9842.94} C_VEL
LIN {X 0,Y 425.851,Z 267.433,A -85,B 0,C 180,E1 -9845.284,E2 -9845.284} C_VEL
LIN {X 0,Y 425.299,Z 264.323,A -85,B 0,C 180,E1 -9846.875,E2 -9846.875} C_VEL
LIN {X 0,Y 425.294,Z 264.324,A -85,B 0,C 180,E1 -9850.128,E2 -9850.128} C_VEL
LIN {X 0,Y 425.266,Z 264.325,A -85,B 0,C 180,E1 -9853.351,E2 -9853.351} C_VEL
LIN {X 0,Y 425.266,Z 264.324,A -85,B 0,C 180,E1 -9856.649,E2 -9856.649} C_VEL
LIN {X 0,Y 425.294,Z 264.323,A -85,B 0,C 180,E1 -9859.872,E2 -9859.872} C_VEL
LIN {X 0,Y 425.285,Z 264.322,A -85,B 0,C 180,E1 -9862.489,E2 -9862.489} C_VEL
LIN {X 0,Y 425.316,Z 264.32,A -85,B 0,C 180,E1 -9865.817,E2 -9865.817} C_VEL
LIN {X 0,Y 425.3,Z 264.322,A -85,B 0,C 180,E1 -9869.238,E2 -9869.238} C_VEL
LIN {X 0,Y 425.358,Z 264.313,A -85,B 0,C 180,E1 -9872.442,E2 -9872.442} C_VEL
LIN {X 0,Y 425.357,Z 264.316,A -85,B 0,C 180,E1 -9875.601,E2 -9875.601} C_VEL
LIN {X 0,Y 425.302,Z 264.32,A -85,B 0,C 180,E1 -9878.681,E2 -9878.681} C_VEL
LIN {X 0,Y 425.33,Z 264.317,A -85,B 0,C 180,E1 -9881.701,E2 -9881.701} C_VEL
LIN {X 0,Y 425.356,Z 264.315,A -85,B 0,C 180,E1 -9884.67,E2 -9884.67} C_VEL
LIN {X 0,Y 425.42,Z 264.306,A -85,B 0,C 180,E1 -9887.597,E2 -9887.597} C_VEL
LIN {X 0,Y 425.415,Z 264.307,A -85,B 0,C 180,E1 -9891.448,E2 -9891.448} C_VEL
LIN {X 0,Y 425.554,Z 264.29,A -85,B 0,C 180,E1 -9894.312,E2 -9894.312} C_VEL
LIN {X 0,Y 425.579,Z 264.287,A -85,B 0,C 180,E1 -9898.106,E2 -9898.106} C_VEL
LIN {X 0,Y 425.707,Z 264.27,A -85,B 0,C 180,E1 -9899.998,E2 -9899.998} C_VEL
LIN {X 0,Y 425.561,Z 264.29,A -85,B 0,C 180,E1 -9902.838,E2 -9902.838} C_VEL
LIN {X 0,Y 425.536,Z 264.294,A -85,B 0,C 180,E1 -9906.637,E2 -9906.637} C_VEL
LIN {X 0,Y 425.405,Z 264.307,A -85,B 0,C 180,E1 -9909.507,E2 -9909.507} C_VEL
LIN {X 0,Y 425.396,Z 264.309,A -85,B 0,C 180,E1 -9912.901,E2 -9912.901} C_VEL
LIN {X 0,Y 425.363,Z 264.314,A -85,B 0,C 180,E1 -9916.603,E2 -9916.603} C_VEL
LIN {X 0,Y 425.329,Z 264.319,A -85,B 0,C 180,E1 -9919.633,E2 -9919.633} C_VEL
LIN {X 0,Y 425.306,Z 264.32,A -85,B 0,C 180,E1 -9923.363,E2 -9923.363} C_VEL
LIN {X 0,Y 425.346,Z 264.314,A -85,B 0,C 180,E1 -9926.842,E2 -9926.842} C_VEL
LIN {X 0,Y 425.288,Z 264.324,A -85,B 0,C 180,E1 -9929.717,E2 -9929.717} C_VEL
LIN {X 0,Y 425.278,Z 264.323,A -85,B 0,C 180,E1 -9933.046,E2 -9933.046} C_VEL
LIN {X 0,Y 425.28,Z 264.325,A -85,B 0,C 180,E1 -9935.927,E2 -9935.927} C_VEL
LIN {X 0,Y 425.306,Z 264.321,A -85,B 0,C 180,E1 -9939.043,E2 -9939.043} C_VEL
LIN {X 0,Y 425.324,Z 264.318,A -85,B 0,C 180,E1 -9942.643,E2 -9942.643} C_VEL
LIN {X 0,Y 425.31,Z 264.319,A -85,B 0,C 180,E1 -9946.049,E2 -9946.049} C_VEL
LIN {X 0,Y 425.301,Z 264.321,A -85,B 0,C 180,E1 -9948.623,E2 -9948.623} C_VEL
LIN {X 0,Y 425.314,Z 264.321,A -85,B 0,C 180,E1 -9951.102,E2 -9951.102} C_VEL
LIN {X 0,Y 425.289,Z 264.324,A -85,B 0,C 180,E1 -9954.662,E2 -9954.662} C_VEL
LIN {X 0,Y 425.253,Z 264.326,A -85,B 0,C 180,E1 -9958.071,E2 -9958.071} C_VEL
LIN {X 0,Y 425.324,Z 264.318,A -85,B 0,C 180,E1 -9961.366,E2 -9961.366} C_VEL
LIN {X 0,Y 425.282,Z 264.325,A -85,B 0,C 180,E1 -9964.553,E2 -9964.553} C_VEL
LIN {X 0,Y 425.307,Z 264.319,A -85,B 0,C 180,E1 -9967.717,E2 -9967.717} C_VEL
LIN {X 0,Y 425.328,Z 264.319,A -85,B 0,C 180,E1 -9970.701,E2 -9970.701} C_VEL
LIN {X 0,Y 425.001,Z 264.358,A -85,B 0,C 180,E1 -9973.672,E2 -9973.672} C_VEL
LIN {X 0,Y 424.84,Z 264.381,A -85,B 0,C 180,E1 -9974.651,E2 -9974.651} C_VEL
LIN {X 0,Y 424.76,Z 264.946,A -85,B 0,C 180,E1 -9975.629,E2 -9975.629} C_VEL
LIN {X 0,Y 424.83,Z 267.315,A -85,B 0,C 180,E1 -9977.58,E2 -9977.58} C_VEL
LIN {X 0,Y 424.679,Z 272.002,A -85,B 0,C 180,E1 -9981.433,E2 -9981.433} C_VEL
LIN {X 0,Y 424.705,Z 274.374,A -85,B 0,C 180,E1 -9983.347,E2 -9983.347} C_VEL
LIN {X 0,Y 424.613,Z 277.955,A -85,B 0,C 180,E1 -9986.203,E2 -9986.203} C_VEL
LIN {X 0,Y 424.292,Z 282.834,A -85,B 0,C 180,E1 -9989.999,E2 -9989.999} C_VEL
LIN {X 0,Y 424.29,Z 284.208,A -85,B 0,C 180,E1 -9990.978,E2 -9990.978} C_VEL
LIN {X 0,Y 426.232,Z 295.414,A -85,B 0,C 180,E1 -9991.475,E2 -9991.475} C_VEL
LIN {X 0,Y 426.866,Z 300.888,A -85,B 0,C 180,E1 -9991.768,E2 -9991.768} C_VEL
LIN {X 0,Y 426.484,Z 311.568,A -85,B 0,C 180,E1 -9992.478,E2 -9992.478} C_VEL
LIN {X 0,Y 426.128,Z 319.914,A -85,B 0,C 180,E1 -9993.19,E2 -9993.19} C_VEL
LIN {X 0,Y 425.714,Z 327.821,A -85,B 0,C 180,E1 -9994.022,E2 -9994.022} C_VEL
LIN {X 0,Y 425.434,Z 335.158,A -85,B 0,C 180,E1 -9994.972,E2 -9994.972} C_VEL
LIN {X 0,Y 424.611,Z 339.166,A -85,B 0,C 180,E1 -9995.551,E2 -9995.551} C_VEL
LIN {X 0,Y 421.464,Z 345.16,A -85,B 0,C 180,E1 -9996.538,E2 -9996.538} C_VEL
LIN {X 0,Y 418.304,Z 350.279,A -85,B 0,C 180,E1 -9997.619,E2 -9997.619} C_VEL
LIN {X 0,Y 417.474,Z 352.899,A -85,B 0,C 180,E1 -9998.34,E2 -9998.34} C_VEL
LIN {X 0,Y 417.265,Z 356.966,A -85,B 0,C 180,E1 -9999.695,E2 -9999.695} C_VEL
LIN {X 0,Y 417.18,Z 359.236,A -85,B 0,C 180,E1 -10000.678,E2 -10000.678} C_VEL
LIN {X 0,Y 417.089,Z 361.56,A -85,B 0,C 180,E1 -10002.243,E2 -10002.243} C_VEL
LIN {X 0,Y 417.009,Z 362.559,A -85,B 0,C 180,E1 -10003.646,E2 -10003.646} C_VEL
LIN {X 0,Y 417.005,Z 362.656,A -85,B 0,C 180,E1 -10004.642,E2 -10004.642} C_VEL
LIN {X 0,Y 417.075,Z 362.255,A -85,B 0,C 180,E1 -10005.64,E2 -10005.64} C_VEL
LIN {X 0,Y 417.168,Z 361.274,A -85,B 0,C 180,E1 -10006.641,E2 -10006.641} C_VEL
LIN {X 0,Y 417.341,Z 358.727,A -85,B 0,C 180,E1 -10008.15,E2 -10008.15} C_VEL
LIN {X 0,Y 417.595,Z 355.169,A -85,B 0,C 180,E1 -10009.539,E2 -10009.539} C_VEL
LIN {X 0,Y 417.832,Z 351.312,A -85,B 0,C 180,E1 -10010.683,E2 -10010.683} C_VEL
LIN {X 0,Y 418.128,Z 347.061,A -85,B 0,C 180,E1 -10011.701,E2 -10011.701} C_VEL
LIN {X 0,Y 418.498,Z 341.877,A -85,B 0,C 180,E1 -10012.72,E2 -10012.72} C_VEL
LIN {X 0,Y 418.913,Z 335.54,A -85,B 0,C 180,E1 -10013.742,E2 -10013.742} C_VEL
LIN {X 0,Y 419.324,Z 328.816,A -85,B 0,C 180,E1 -10014.638,E2 -10014.638} C_VEL
LIN {X 0,Y 419.785,Z 321.556,A -85,B 0,C 180,E1 -10015.438,E2 -10015.438} C_VEL
LIN {X 0,Y 420.287,Z 313.412,A -85,B 0,C 180,E1 -10016.169,E2 -10016.169} C_VEL
LIN {X 0,Y 420.716,Z 304.47,A -85,B 0,C 180,E1 -10016.808,E2 -10016.808} C_VEL
LIN {X 0,Y 420.642,Z 300.859,A -85,B 0,C 180,E1 -10017.041,E2 -10017.041} C_VEL
LIN {X 0,Y 418.55,Z 290.354,A -85,B 0,C 180,E1 -10017.633,E2 -10017.633} C_VEL
LIN {X 0,Y 417.262,Z 284.671,A -85,B 0,C 180,E1 -10017.918,E2 -10017.918} C_VEL
LIN {X 0,Y 417.373,Z 281.127,A -85,B 0,C 180,E1 -10020.826,E2 -10020.826} C_VEL
LIN {X 0,Y 417.402,Z 277.641,A -85,B 0,C 180,E1 -10023.753,E2 -10023.753} C_VEL
LIN {X 0,Y 417.56,Z 273.494,A -85,B 0,C 180,E1 -10027.293,E2 -10027.293} C_VEL
LIN {X 0,Y 417.711,Z 269.491,A -85,B 0,C 180,E1 -10030.793,E2 -10030.793} C_VEL
LIN {X 0,Y 417.86,Z 266.274,A -85,B 0,C 180,E1 -10033.683,E2 -10033.683} C_VEL
LIN {X 0,Y 417.944,Z 265.238,A -85,B 0,C 180,E1 -10035.072,E2 -10035.072} C_VEL
LIN {X 0,Y 418.153,Z 265.212,A -85,B 0,C 180,E1 -10037.759,E2 -10037.759} C_VEL
LIN {X 0,Y 418.248,Z 265.199,A -85,B 0,C 180,E1 -10040.618,E2 -10040.618} C_VEL
LIN {X 0,Y 418.227,Z 265.205,A -85,B 0,C 180,E1 -10043.977,E2 -10043.977} C_VEL
LIN {X 0,Y 418.238,Z 265.202,A -85,B 0,C 180,E1 -10047.157,E2 -10047.157} C_VEL
LIN {X 0,Y 418.25,Z 265.199,A -85,B 0,C 180,E1 -10050.897,E2 -10050.897} C_VEL
LIN {X 0,Y 418.251,Z 265.199,A -85,B 0,C 180,E1 -10054.097,E2 -10054.097} C_VEL
LIN {X 0,Y 418.215,Z 265.204,A -85,B 0,C 180,E1 -10057.265,E2 -10057.265} C_VEL
LIN {X 0,Y 418.267,Z 265.198,A -85,B 0,C 180,E1 -10060.366,E2 -10060.366} C_VEL
LIN {X 0,Y 418.301,Z 265.195,A -85,B 0,C 180,E1 -10063.406,E2 -10063.406} C_VEL
LIN {X 0,Y 418.341,Z 265.187,A -85,B 0,C 180,E1 -10066.995,E2 -10066.995} C_VEL
LIN {X 0,Y 418.347,Z 265.184,A -85,B 0,C 180,E1 -10070.331,E2 -10070.331} C_VEL
LIN {X 0,Y 418.445,Z 265.17,A -85,B 0,C 180,E1 -10073.25,E2 -10073.25} C_VEL
LIN {X 0,Y 418.327,Z 265.188,A -85,B 0,C 180,E1 -10075.183,E2 -10075.183} C_VEL
LIN {X 0,Y 418.534,Z 265.16,A -85,B 0,C 180,E1 -10078.077,E2 -10078.077} C_VEL
LIN {X 0,Y 418.66,Z 265.147,A -85,B 0,C 180,E1 -10080.002,E2 -10080.002} C_VEL
LIN {X 0,Y 418.49,Z 265.167,A -85,B 0,C 180,E1 -10082.89,E2 -10082.89} C_VEL
LIN {X 0,Y 418.484,Z 265.167,A -85,B 0,C 180,E1 -10086.753,E2 -10086.753} C_VEL
LIN {X 0,Y 418.332,Z 265.188,A -85,B 0,C 180,E1 -10089.673,E2 -10089.673} C_VEL
LIN {X 0,Y 418.346,Z 265.187,A -85,B 0,C 180,E1 -10093.008,E2 -10093.008} C_VEL
LIN {X 0,Y 418.304,Z 265.194,A -85,B 0,C 180,E1 -10096.737,E2 -10096.737} C_VEL
LIN {X 0,Y 418.262,Z 265.199,A -85,B 0,C 180,E1 -10099.792,E2 -10099.792} C_VEL
LIN {X 0,Y 418.225,Z 265.204,A -85,B 0,C 180,E1 -10102.738,E2 -10102.738} C_VEL
LIN {X 0,Y 418.231,Z 265.205,A -85,B 0,C 180,E1 -10105.908,E2 -10105.908} C_VEL
LIN {X 0,Y 418.254,Z 265.204,A -85,B 0,C 180,E1 -10109.164,E2 -10109.164} C_VEL
LIN {X 0,Y 418.252,Z 265.202,A -85,B 0,C 180,E1 -10112.846,E2 -10112.846} C_VEL
LIN {X 0,Y 418.239,Z 265.202,A -85,B 0,C 180,E1 -10116.239,E2 -10116.239} C_VEL
LIN {X 0,Y 418.259,Z 265.198,A -85,B 0,C 180,E1 -10119.682,E2 -10119.682} C_VEL
LIN {X 0,Y 418.241,Z 265.201,A -85,B 0,C 180,E1 -10122.325,E2 -10122.325} C_VEL
LIN {X 0,Y 418.232,Z 265.206,A -85,B 0,C 180,E1 -10125.11,E2 -10125.11} C_VEL
LIN {X 0,Y 418.236,Z 265.206,A -85,B 0,C 180,E1 -10127.769,E2 -10127.769} C_VEL
LIN {X 0,Y 418.282,Z 265.209,A -85,B 0,C 180,E1 -10131.101,E2 -10131.101} C_VEL
LIN {X 0,Y 419.371,Z 271.605,A -85,B 0,C 180,E1 -10134.672,E2 -10134.672} C_VEL
LIN {X 0,Y 419.913,Z 275.714,A -85,B 0,C 180,E1 -10136.809,E2 -10136.809} C_VEL
LIN {X 0,Y 419.527,Z 280.803,A -85,B 0,C 180,E1 -10139.275,E2 -10139.275} C_VEL
LIN {X 0,Y 418.997,Z 286.662,A -85,B 0,C 180,E1 -10141.99,E2 -10141.99} C_VEL
LIN {X 0,Y 418.395,Z 294.945,A -85,B 0,C 180,E1 -10145.7,E2 -10145.7} C_VEL
LIN {X 0,Y 417.883,Z 303.296,A -85,B 0,C 180,E1 -10149.32,E2 -10149.32} C_VEL
LIN {X 0,Y 417.579,Z 311.739,A -85,B 0,C 180,E1 -10152.872,E2 -10152.872} C_VEL
LIN {X 0,Y 417.314,Z 319.504,A -85,B 0,C 180,E1 -10156.085,E2 -10156.085} C_VEL
LIN {X 0,Y 419.186,Z 333.013,A -85,B 0,C 180,E1 -10156.682,E2 -10156.682} C_VEL
LIN {X 0,Y 419.827,Z 342.244,A -85,B 0,C 180,E1 -10157.222,E2 -10157.222} C_VEL
LIN {X 0,Y 419.708,Z 350.335,A -85,B 0,C 180,E1 -10157.797,E2 -10157.797} C_VEL
LIN {X 0,Y 419.132,Z 358.62,A -85,B 0,C 180,E1 -10158.516,E2 -10158.516} C_VEL
LIN {X 0,Y 418.643,Z 366.477,A -85,B 0,C 180,E1 -10159.36,E2 -10159.36} C_VEL
LIN {X 0,Y 418.185,Z 373.838,A -85,B 0,C 180,E1 -10160.326,E2 -10160.326} C_VEL
LIN {X 0,Y 417.731,Z 381.323,A -85,B 0,C 180,E1 -10161.536,E2 -10161.536} C_VEL
LIN {X 0,Y 417.383,Z 387.219,A -85,B 0,C 180,E1 -10162.746,E2 -10162.746} C_VEL
LIN {X 0,Y 417.174,Z 392.64,A -85,B 0,C 180,E1 -10164.2,E2 -10164.2} C_VEL
LIN {X 0,Y 417.091,Z 396.673,A -85,B 0,C 180,E1 -10165.653,E2 -10165.653} C_VEL
LIN {X 0,Y 417.088,Z 399.456,A -85,B 0,C 180,E1 -10167.104,E2 -10167.104} C_VEL
LIN {X 0,Y 417.094,Z 400.584,A -85,B 0,C 180,E1 -10168.07,E2 -10168.07} C_VEL
LIN {X 0,Y 417.056,Z 401.24,A -85,B 0,C 180,E1 -10169.036,E2 -10169.036} C_VEL
LIN {X 0,Y 417.054,Z 401.436,A -85,B 0,C 180,E1 -10170.001,E2 -10170.001} C_VEL
LIN {X 0,Y 417.056,Z 401.114,A -85,B 0,C 180,E1 -10170.967,E2 -10170.967} C_VEL
LIN {X 0,Y 417.096,Z 400.207,A -85,B 0,C 180,E1 -10171.932,E2 -10171.932} C_VEL
LIN {X 0,Y 417.122,Z 398.81,A -85,B 0,C 180,E1 -10172.899,E2 -10172.899} C_VEL
LIN {X 0,Y 417.092,Z 395.739,A -85,B 0,C 180,E1 -10174.35,E2 -10174.35} C_VEL
LIN {X 0,Y 417.159,Z 391.35,A -85,B 0,C 180,E1 -10175.803,E2 -10175.803} C_VEL
LIN {X 0,Y 417.454,Z 385.266,A -85,B 0,C 180,E1 -10177.255,E2 -10177.255} C_VEL
LIN {X 0,Y 417.592,Z 380.222,A -85,B 0,C 180,E1 -10178.226,E2 -10178.226} C_VEL
LIN {X 0,Y 417.87,Z 374.147,A -85,B 0,C 180,E1 -10179.195,E2 -10179.195} C_VEL
LIN {X 0,Y 418.252,Z 366.754,A -85,B 0,C 180,E1 -10180.163,E2 -10180.163} C_VEL
LIN {X 0,Y 418.622,Z 358.832,A -85,B 0,C 180,E1 -10181.01,E2 -10181.01} C_VEL
LIN {X 0,Y 419.089,Z 350.473,A -85,B 0,C 180,E1 -10181.733,E2 -10181.733} C_VEL
LIN {X 0,Y 419.235,Z 341.681,A -85,B 0,C 180,E1 -10182.343,E2 -10182.343} C_VEL
LIN {X 0,Y 418.218,Z 329.289,A -85,B 0,C 180,E1 -10182.997,E2 -10182.997} C_VEL
LIN {X 0,Y 417.216,Z 319.852,A -85,B 0,C 180,E1 -10183.348,E2 -10183.348} C_VEL
LIN {X 0,Y 417.464,Z 311.737,A -85,B 0,C 180,E1 -10186.631,E2 -10186.631} C_VEL
LIN {X 0,Y 417.728,Z 303.075,A -85,B 0,C 180,E1 -10190.177,E2 -10190.177} C_VEL
LIN {X 0,Y 418.12,Z 295.646,A -85,B 0,C 180,E1 -10193.267,E2 -10193.267} C_VEL
LIN {X 0,Y 418.575,Z 286.961,A -85,B 0,C 180,E1 -10196.959,E2 -10196.959} C_VEL
LIN {X 0,Y 419.127,Z 279.548,A -85,B 0,C 180,E1 -10200.203,E2 -10200.203} C_VEL
LIN {X 0,Y 419.489,Z 273.12,A -85,B 0,C 180,E1 -10203.102,E2 -10203.102} C_VEL
LIN {X 0,Y 418.821,Z 268.388,A -85,B 0,C 180,E1 -10205.376,E2 -10205.376} C_VEL
LIN {X 0,Y 418.258,Z 265.2,A -85,B 0,C 180,E1 -10206.969,E2 -10206.969} C_VEL
LIN {X 0,Y 418.253,Z 265.2,A -85,B 0,C 180,E1 -10209.683,E2 -10209.683} C_VEL
LIN {X 0,Y 418.238,Z 265.202,A -85,B 0,C 180,E1 -10212.321,E2 -10212.321} C_VEL
LIN {X 0,Y 418.244,Z 265.198,A -85,B 0,C 180,E1 -10215.109,E2 -10215.109} C_VEL
LIN {X 0,Y 418.249,Z 265.201,A -85,B 0,C 180,E1 -10217.767,E2 -10217.767} C_VEL
LIN {X 0,Y 418.251,Z 265.198,A -85,B 0,C 180,E1 -10220.621,E2 -10220.621} C_VEL
LIN {X 0,Y 418.251,Z 265.2,A -85,B 0,C 180,E1 -10223.975,E2 -10223.975} C_VEL
LIN {X 0,Y 418.267,Z 265.198,A -85,B 0,C 180,E1 -10227.156,E2 -10227.156} C_VEL
LIN {X 0,Y 418.278,Z 265.196,A -85,B 0,C 180,E1 -10230.895,E2 -10230.895} C_VEL
LIN {X 0,Y 418.277,Z 265.195,A -85,B 0,C 180,E1 -10234.095,E2 -10234.095} C_VEL
LIN {X 0,Y 418.241,Z 265.202,A -85,B 0,C 180,E1 -10237.263,E2 -10237.263} C_VEL
LIN {X 0,Y 418.292,Z 265.192,A -85,B 0,C 180,E1 -10240.363,E2 -10240.363} C_VEL
LIN {X 0,Y 418.325,Z 265.192,A -85,B 0,C 180,E1 -10243.404,E2 -10243.404} C_VEL
LIN {X 0,Y 418.355,Z 265.188,A -85,B 0,C 180,E1 -10246.998,E2 -10246.998} C_VEL
LIN {X 0,Y 418.346,Z 265.187,A -85,B 0,C 180,E1 -10250.327,E2 -10250.327} C_VEL
LIN {X 0,Y 418.479,Z 265.171,A -85,B 0,C 180,E1 -10253.247,E2 -10253.247} C_VEL
LIN {X 0,Y 418.343,Z 265.188,A -85,B 0,C 180,E1 -10255.18,E2 -10255.18} C_VEL
LIN {X 0,Y 418.548,Z 265.162,A -85,B 0,C 180,E1 -10258.074,E2 -10258.074} C_VEL
LIN {X 0,Y 418.677,Z 265.146,A -85,B 0,C 180,E1 -10259.998,E2 -10259.998} C_VEL
LIN {X 0,Y 418.515,Z 265.167,A -85,B 0,C 180,E1 -10262.886,E2 -10262.886} C_VEL
LIN {X 0,Y 418.498,Z 265.17,A -85,B 0,C 180,E1 -10266.749,E2 -10266.749} C_VEL
LIN {X 0,Y 418.404,Z 265.182,A -85,B 0,C 180,E1 -10268.693,E2 -10268.693} C_VEL
LIN {X 0,Y 418.318,Z 265.19,A -85,B 0,C 180,E1 -10271.629,E2 -10271.629} C_VEL
LIN {X 0,Y 418.305,Z 265.193,A -85,B 0,C 180,E1 -10274.595,E2 -10274.595} C_VEL
LIN {X 0,Y 418.29,Z 265.195,A -85,B 0,C 180,E1 -10277.602,E2 -10277.602} C_VEL
LIN {X 0,Y 418.25,Z 265.199,A -85,B 0,C 180,E1 -10280.661,E2 -10280.661} C_VEL
LIN {X 0,Y 418.287,Z 265.196,A -85,B 0,C 180,E1 -10283.779,E2 -10283.779} C_VEL
LIN {X 0,Y 418.308,Z 265.191,A -85,B 0,C 180,E1 -10287.068,E2 -10287.068} C_VEL
LIN {X 0,Y 418.242,Z 265.2,A -85,B 0,C 180,E1 -10290.27,E2 -10290.27} C_VEL
LIN {X 0,Y 418.245,Z 265.202,A -85,B 0,C 180,E1 -10293.675,E2 -10293.675} C_VEL
LIN {X 0,Y 418.241,Z 265.201,A -85,B 0,C 180,E1 -10297.221,E2 -10297.221} C_VEL
LIN {X 0,Y 418.259,Z 265.199,A -85,B 0,C 180,E1 -10299.678,E2 -10299.678} C_VEL
LIN {X 0,Y 418.278,Z 265.195,A -85,B 0,C 180,E1 -10302.327,E2 -10302.327} C_VEL
LIN {X 0,Y 418.266,Z 265.199,A -85,B 0,C 180,E1 -10305.112,E2 -10305.112} C_VEL
LIN {X 0,Y 418.283,Z 265.195,A -85,B 0,C 180,E1 -10307.771,E2 -10307.771} C_VEL
LIN {X 0,Y 418.256,Z 265.198,A -85,B 0,C 180,E1 -10311.557,E2 -10311.557} C_VEL
LIN {X 0,Y 418.248,Z 265.201,A -85,B 0,C 180,E1 -10315.157,E2 -10315.157} C_VEL
LIN {X 0,Y 418.233,Z 265.201,A -85,B 0,C 180,E1 -10317.47,E2 -10317.47} C_VEL
LIN {X 0,Y 418.263,Z 265.199,A -85,B 0,C 180,E1 -10320.891,E2 -10320.891} C_VEL
LIN {X 0,Y 418.257,Z 265.198,A -85,B 0,C 180,E1 -10324.094,E2 -10324.094} C_VEL
LIN {X 0,Y 418.26,Z 265.197,A -85,B 0,C 180,E1 -10327.535,E2 -10327.535} C_VEL
LIN {X 0,Y 418.261,Z 265.199,A -85,B 0,C 180,E1 -10330.362,E2 -10330.362} C_VEL
LIN {X 0,Y 417.999,Z 265.23,A -85,B 0,C 180,E1 -10333.399,E2 -10333.399} C_VEL
LIN {X 0,Y 417.711,Z 265.38,A -85,B 0,C 180,E1 -10335.381,E2 -10335.381} C_VEL
LIN {X 0,Y 417.713,Z 268.932,A -85,B 0,C 180,E1 -10338.351,E2 -10338.351} C_VEL
LIN {X 0,Y 417.62,Z 273.679,A -85,B 0,C 180,E1 -10342.262,E2 -10342.262} C_VEL
LIN {X 0,Y 417.567,Z 277.264,A -85,B 0,C 180,E1 -10345.171,E2 -10345.171} C_VEL
LIN {X 0,Y 417.509,Z 279.692,A -85,B 0,C 180,E1 -10347.104,E2 -10347.104} C_VEL
LIN {X 0,Y 417.222,Z 284.374,A -85,B 0,C 180,E1 -10350.783,E2 -10350.783} C_VEL
LIN {X 0,Y 419.23,Z 296.1,A -85,B 0,C 180,E1 -10351.32,E2 -10351.32} C_VEL
LIN {X 0,Y 419.877,Z 301.517,A -85,B 0,C 180,E1 -10351.617,E2 -10351.617} C_VEL
LIN {X 0,Y 419.513,Z 311.362,A -85,B 0,C 180,E1 -10352.279,E2 -10352.279} C_VEL
LIN {X 0,Y 419.145,Z 319.801,A -85,B 0,C 180,E1 -10353.002,E2 -10353.002} C_VEL
LIN {X 0,Y 418.702,Z 327.786,A -85,B 0,C 180,E1 -10353.848,E2 -10353.848} C_VEL
LIN {X 0,Y 418.467,Z 333.499,A -85,B 0,C 180,E1 -10354.574,E2 -10354.574} C_VEL
LIN {X 0,Y 418.096,Z 339.9,A -85,B 0,C 180,E1 -10355.545,E2 -10355.545} C_VEL
LIN {X 0,Y 417.945,Z 345.193,A -85,B 0,C 180,E1 -10356.516,E2 -10356.516} C_VEL
LIN {X 0,Y 417.754,Z 348.818,A -85,B 0,C 180,E1 -10357.284,E2 -10357.284} C_VEL
LIN {X 0,Y 417.474,Z 352.899,A -85,B 0,C 180,E1 -10358.34,E2 -10358.34} C_VEL
LIN {X 0,Y 416.686,Z 355.332,A -85,B 0,C 180,E1 -10359.079,E2 -10359.079} C_VEL
LIN {X 0,Y 413.694,Z 358.603,A -85,B 0,C 180,E1 -10360.303,E2 -10360.303} C_VEL
LIN {X 0,Y 411.205,Z 360.619,A -85,B 0,C 180,E1 -10361.314,E2 -10361.314} C_VEL
LIN {X 0,Y 410.106,Z 361.76,A -85,B 0,C 180,E1 -10362.112,E2 -10362.112} C_VEL
